SMOVL C00195 BC00195 V=166.7  +MOVJ EC00195
SFTOF3D
MOVL C00196 BC00196 V=1000.0  +MOVJ EC00196 VJ=100.00
'EndPath S3470
'Path S4850
SFTOF3D
MOVL C00197 BC00197 V=666.7  +MOVJ EC00197 VJ=100.00
SMOVL C00198 BC00198 V=166.7  +MOVJ EC00198
SREFP 3 C00199 BC00199  +REFP EC00199
CALL JOB:SEARCH-R1-S13D
SET P071 P006
SFTON3D P071
SMOVL C00200 BC00200 V=166.7  +MOVJ EC00200
SREFP 3 C00201 BC00201  +REFP EC00201
CALL JOB:SEARCH-R1-S13D
SET P071 P006
SFTON3D P071
SMOVL C00202 BC00202 V=166.7  +MOVJ EC00202
SMOVL C00203 BC00203 V=166.7  +MOVJ EC00203
SREFP 3 C00204 BC00204  +REFP EC00204
CALL JOB:SEARCH-R1-S13D
SET P071 P006
SFTON3D P071
SMOVL C00205 BC00205 V=166.7  +MOVJ EC00205
MOVL C00206 BC00206 V=1000.0  +MOVJ EC00206 VJ=100.00
'EndPath S4850
'Path S4851
SFTOF3D
MOVJ C00207 BC00207 VJ=100.00  +MOVJ EC00207 VJ=100.00
'POMIAR_DOD_WZM_BOK
MOVL C00208 BC00208 V=666.7  +MOVJ EC00208 VJ=100.00
SMOVL C00209 BC00209 V=166.7  +MOVJ EC00209
SREFP 3 C00210 BC00210  +REFP EC00210
CALL JOB:SEARCH-R1-S13D
SET P080 P006
SFTON3D P080
SMOVL C00211 BC00211 V=166.7  +MOVJ EC00211
SREFP 3 C00212 BC00212  +REFP EC00212
CALL JOB:SEARCH-R1-S13D
SET P080 P006
SFTON3D P080
SMOVL C00213 BC00213 V=166.7  +MOVJ EC00213
MOVL C00214 BC00214 V=666.7  +MOVJ EC00214 VJ=100.00
SMOVL C00215 BC00215 V=166.7  +MOVJ EC00215
SREFP 3 C00216 BC00216  +REFP EC00216
CALL JOB:SEARCH-R1-S13D
SET P042 P006
SFTON3D P042
SMOVL C00217 BC00217 V=166.7  +MOVJ EC00217
SREFP 3 C00218 BC00218  +REFP EC00218
CALL JOB:SEARCH-R1-S13D
SET P042 P006
SFTON3D P042
SMOVL C00219 BC00219 V=166.7  +MOVJ EC00219
SREFP 3 C00220 BC00220  +REFP EC00220
CALL JOB:SEARCH-R1-S13D
SET P043 P006
SFTON3D P043
SMOVL C00221 BC00221 V=166.7  +MOVJ EC00221
SREFP 3 C00222 BC00222  +REFP EC00222
CALL JOB:SEARCH-R1-S13D
SET P043 P006
SFTON3D P043
SMOVL C00223 BC00223 V=166.7  +MOVJ EC00223
SMOVL C00224 BC00224 V=1000.0  +MOVJ EC00224
MOVL C00225 BC00225 V=666.7  +MOVJ EC00225 VJ=100.00
SMOVL C00226 BC00226 V=166.7  +MOVJ EC00226
SREFP 3 C00227 BC00227  +REFP EC00227
CALL JOB:SEARCH-R1-S13D
SET P044 P006
SFTON3D P044
SMOVL C00228 BC00228 V=166.7  +MOVJ EC00228
SREFP 3 C00229 BC00229  +REFP EC00229
CALL JOB:SEARCH-R1-S13D
SET P044 P006
SFTON3D P044
SMOVL C00230 BC00230 V=166.7  +MOVJ EC00230
MOVL C00231 BC00231 V=666.7  +MOVJ EC00231 VJ=100.00
SMOVL C00232 BC00232 V=166.7  +MOVJ EC00232
SREFP 3 C00233 BC00233  +REFP EC00233
CALL JOB:SEARCH-R1-S13D
SET P045 P006
SFTON3D P045
SMOVL C00234 BC00234 V=166.7  +MOVJ EC00234
SREFP 3 C00235 BC00235  +REFP EC00235
CALL JOB:SEARCH-R1-S13D
SET P045 P006
SFTON3D P045
SMOVL C00236 BC00236 V=166.7  +MOVJ EC00236
SREFP 3 C00237 BC00237  +REFP EC00237
CALL JOB:SEARCH-R1-S13D
SET P046 P006
SFTON3D P046
SMOVL C00238 BC00238 V=166.7  +MOVJ EC00238
SREFP 3 C00239 BC00239  +REFP EC00239
CALL JOB:SEARCH-R1-S13D
SET P046 P006
SFTON3D P046
SMOVL C00240 BC00240 V=166.7  +MOVJ EC00240
SFTOF3D
SFTOF3D
MOVJ C00241 BC00241 VJ=100.00  +MOVJ EC00241 VJ=100.00
MOVL C00242 BC00242 V=666.7  +MOVJ EC00242 VJ=100.00
MOVL C00243 BC00243 V=1000.0  +MOVJ EC00243 VJ=0.78
SMOVL C00244 BC00244 V=166.7  +MOVJ EC00244
SREFP 3 C00245 BC00245  +REFP EC00245
CALL JOB:SEARCH-R1-S13D
SET P072 P006
SFTON3D P072
SMOVL C00246 BC00246 V=166.7  +MOVJ EC00246
SREFP 3 C00247 BC00247  +REFP EC00247
CALL JOB:SEARCH-R1-S13D
SET P072 P006
SFTON3D P072
SMOVL C00248 BC00248 V=166.7  +MOVJ EC00248
SMOVL C00249 BC00249 V=166.7  +MOVJ EC00249
SREFP 3 C00250 BC00250  +REFP EC00250
CALL JOB:SEARCH-R1-S13D
SET P072 P006
SFTON3D P072
SMOVL C00251 BC00251 V=166.7  +MOVJ EC00251
SFTOF3D
MOVL C00252 BC00252 V=1000.0  +MOVJ EC00252 VJ=100.00
'EndPath S4851
MOVJ C00253 BC00253 VJ=100.00  +MOVJ EC00253 VJ=100.00
MOVJ C00254 BC00254 VJ=100.00  +MOVJ EC00254 VJ=100.00
'Path S4852
SFTOF3D
MOVJ C00255 BC00255 VJ=100.00  +MOVJ EC00255 VJ=100.00
MOVL C00256 BC00256 V=666.7  +MOVJ EC00256 VJ=100.00
SMOVL C00257 BC00257 V=166.7  +MOVJ EC00257
SREFP 3 C00258 BC00258  +REFP EC00258
CALL JOB:SEARCH-R1-S13D
SET P073 P006
SFTON3D P073
SMOVL C00259 BC00259 V=166.7  +MOVJ EC00259
SMOVL C00260 BC00260 V=166.7  +MOVJ EC00260
SREFP 3 C00261 BC00261  +REFP EC00261
CALL JOB:SEARCH-R1-S13D
SET P073 P006
SFTON3D P073
SMOVL C00262 BC00262 V=166.7  +MOVJ EC00262
SMOVL C00263 BC00263 V=166.7  +MOVJ EC00263
SREFP 3 C00264 BC00264  +REFP EC00264
CALL JOB:SEARCH-R1-S13D
SET P073 P006
SFTON3D P073
SMOVL C00265 BC00265 V=166.7  +MOVJ EC00265
MOVL C00266 BC00266 V=1000.0  +MOVJ EC00266 VJ=100.00
'EndPath S4852
MOVJ C00267 BC00267 VJ=100.00  +MOVJ EC00267 VJ=100.00
'Path S4853
SFTOF3D
MOVJ C00268 BC00268 VJ=100.00  +MOVJ EC00268 VJ=100.00
MOVL C00269 BC00269 V=666.7  +MOVJ EC00269 VJ=100.00
SMOVL C00270 BC00270 V=166.7  +MOVJ EC00270
SREFP 3 C00271 BC00271  +REFP EC00271
CALL JOB:SEARCH-R1-S13D
SET P074 P006
SFTON3D P074
SMOVL C00272 BC00272 V=166.7  +MOVJ EC00272
SMOVL C00273 BC00273 V=333.3  +MOVJ EC00273
SREFP 3 C00274 BC00274  +REFP EC00274
CALL JOB:SEARCH-R1-S13D
SET P074 P006
SFTON3D P074
SMOVL C00275 BC00275 V=166.7  +MOVJ EC00275
SREFP 3 C00276 BC00276  +REFP EC00276
CALL JOB:SEARCH-R1-S13D
SET P074 P006
SFTON3D P074
SMOVL C00277 BC00277 V=166.7  +MOVJ EC00277
SFTOF3D
MOVL C00278 BC00278 V=1000.0  +MOVJ EC00278 VJ=100.00
'EndPath S4853
'Path S3467
SFTOF3D
MOVJ C00279 BC00279 VJ=100.00  +MOVJ EC00279 VJ=100.00
MOVJ C00280 BC00280 VJ=100.00  +MOVJ EC00280 VJ=100.00
MOVL C00281 BC00281 V=666.7  +MOVJ EC00281 VJ=100.00
SMOVL C00282 BC00282 V=166.7  +MOVJ EC00282
SREFP 3 C00283 BC00283  +REFP EC00283
CALL JOB:SEARCH-R1-S13D
SET P081 P006
SFTON3D P081
SMOVL C00284 BC00284 V=166.7  +MOVJ EC00284
SMOVL C00285 BC00285 V=166.7  +MOVJ EC00285
SREFP 3 C00286 BC00286  +REFP EC00286
CALL JOB:SEARCH-R1-S13D
SET P081 P006
SFTON3D P081
SMOVL C00287 BC00287 V=166.7  +MOVJ EC00287
SMOVL C00288 BC00288 V=800.0  +MOVJ EC00288
SMOVL C00289 BC00289 V=166.7  +MOVJ EC00289
SREFP 3 C00290 BC00290  +REFP EC00290
CALL JOB:SEARCH-R1-S13D
SET P081 P006
SFTON3D P081
SMOVL C00291 BC00291 V=166.7  +MOVJ EC00291
MOVJ C00292 BC00292 VJ=100.00  +MOVJ EC00292 VJ=100.00
MOVJ C00293 BC00293 VJ=100.00  +MOVJ EC00293 VJ=100.00
SFTOF3D
MOVJ C00294 BC00294 VJ=100.00  +MOVJ EC00294 VJ=100.00
MOVL C00295 BC00295 V=666.7  +MOVJ EC00295 VJ=100.00
SMOVL C00296 BC00296 V=166.7  +MOVJ EC00296
SREFP 3 C00297 BC00297  +REFP EC00297
CALL JOB:SEARCH-R1-S13D
SET P026 P006
SFTON3D P026
SMOVL C00298 BC00298 V=166.7  +MOVJ EC00298
SREFP 3 C00299 BC00299  +REFP EC00299
CALL JOB:SEARCH-R1-S13D
SET P026 P006
SFTON3D P026
SMOVL C00300 BC00300 V=166.7  +MOVJ EC00300
SMOVL C00301 BC00301 V=800.0  +MOVJ EC00301
SMOVL C00302 BC00302 V=166.7  +MOVJ EC00302
SREFP 3 C00303 BC00303  +REFP EC00303
CALL JOB:SEARCH-R1-S13D
SET P026 P006
SFTON3D P026
SMOVL C00304 BC00304 V=166.7  +MOVJ EC00304
MOVL C00305 BC00305 V=1000.0  +MOVJ EC00305 VJ=100.00
'EndPath S3467
MOVJ C00306 BC00306 VJ=100.00  +MOVJ EC00306 VJ=100.00
'Path S3466
SFTOF3D
MOVJ C00307 BC00307 VJ=100.00  +MOVJ EC00307 VJ=100.00
MOVL C00308 BC00308 V=666.7  +MOVJ EC00308 VJ=100.00
SMOVL C00309 BC00309 V=166.7  +MOVJ EC00309
SREFP 3 C00310 BC00310  +REFP EC00310
CALL JOB:SEARCH-R1-S13D
SET P025 P006
SFTON3D P025
SMOVL C00311 BC00311 V=166.7  +MOVJ EC00311
SMOVL C00312 BC00312 V=166.7  +MOVJ EC00312
SREFP 3 C00313 BC00313  +REFP EC00313
CALL JOB:SEARCH-R1-S13D
SET P025 P006
SFTON3D P025
SMOVL C00314 BC00314 V=166.7  +MOVJ EC00314
SMOVL C00315 BC00315 V=200.0  +MOVJ EC00315
SMOVL C00316 BC00316 V=166.7  +MOVJ EC00316
SREFP 3 C00317 BC00317  +REFP EC00317
CALL JOB:SEARCH-R1-S13D
SET P025 P006
SFTON3D P025
SMOVL C00318 BC00318 V=166.7  +MOVJ EC00318
MOVL C00319 BC00319 V=1000.0  +MOVJ EC00319 VJ=100.00
MOVL C00320 BC00320 V=1000.0  +MOVJ EC00320 VJ=0.78
SMOVL C00321 BC00321 V=166.7  +MOVJ EC00321
SREFP 3 C00322 BC00322  +REFP EC00322
CALL JOB:SEARCH-R1-S13D
SET P047 P006
SFTON3D P047
SMOVL C00323 BC00323 V=166.7  +MOVJ EC00323
SMOVL C00324 BC00324 V=166.7  +MOVJ EC00324
SREFP 3 C00325 BC00325  +REFP EC00325
CALL JOB:SEARCH-R1-S13D
SET P047 P006
SFTON3D P047
SMOVL C00326 BC00326 V=166.7  +MOVJ EC00326
MOVL C00327 BC00327 V=1000.0  +MOVJ EC00327 VJ=0.78
SMOVL C00328 BC00328 V=166.7  +MOVJ EC00328
SREFP 3 C00329 BC00329  +REFP EC00329
CALL JOB:SEARCH-R1-S13D
SET P048 P006
SFTON3D P048
SMOVL C00330 BC00330 V=166.7  +MOVJ EC00330
SMOVL C00331 BC00331 V=166.7  +MOVJ EC00331
SREFP 3 C00332 BC00332  +REFP EC00332
CALL JOB:SEARCH-R1-S13D
SET P048 P006
SFTON3D P048
SMOVL C00333 BC00333 V=166.7  +MOVJ EC00333
SFTOF3D
MOVL C00334 BC00334 V=1000.0  +MOVJ EC00334 VJ=0.78
'EndPath S3466
MOVJ C00335 BC00335 VJ=100.00  +MOVJ EC00335 VJ=100.00
'Path S3469
SFTOF3D
MOVJ C00336 BC00336 VJ=100.00  +MOVJ EC00336 VJ=100.00
MOVL C00337 BC00337 V=666.7  +MOVJ EC00337 VJ=100.00
SMOVL C00338 BC00338 V=166.7  +MOVJ EC00338
SREFP 3 C00339 BC00339  +REFP EC00339
CALL JOB:SEARCH-R1-S13D
SET P055 P006
SFTON3D P055
SMOVL C00340 BC00340 V=166.7  +MOVJ EC00340
SREFP 3 C00341 BC00341  +REFP EC00341
CALL JOB:SEARCH-R1-S13D
SET P055 P006
SFTON3D P055
SMOVL C00342 BC00342 V=166.7  +MOVJ EC00342
MOVL C00343 BC00343 V=666.7  +MOVJ EC00343 VJ=100.00
SMOVL C00344 BC00344 V=166.7  +MOVJ EC00344
SREFP 3 C00345 BC00345  +REFP EC00345
CALL JOB:SEARCH-R1-S13D
SET P049 P006
SFTON3D P049
SMOVL C00346 BC00346 V=166.7  +MOVJ EC00346
SREFP 3 C00347 BC00347  +REFP EC00347
CALL JOB:SEARCH-R1-S13D
SET P049 P006
SFTON3D P049
SMOVL C00348 BC00348 V=166.7  +MOVJ EC00348
MOVL C00349 BC00349 V=666.7  +MOVJ EC00349 VJ=100.00
SMOVL C00350 BC00350 V=166.7  +MOVJ EC00350
SREFP 3 C00351 BC00351  +REFP EC00351
CALL JOB:SEARCH-R1-S13D
SET P028 P006
SFTON3D P028
SMOVL C00352 BC00352 V=166.7  +MOVJ EC00352
SREFP 3 C00353 BC00353  +REFP EC00353
CALL JOB:SEARCH-R1-S13D
SET P028 P006
SFTON3D P028
SMOVL C00354 BC00354 V=166.7  +MOVJ EC00354
SMOVL C00355 BC00355 V=333.3  +MOVJ EC00355
SMOVL C00356 BC00356 V=166.7  +MOVJ EC00356
SREFP 3 C00357 BC00357  +REFP EC00357
CALL JOB:SEARCH-R1-S13D
SET P028 P006
SFTON3D P028
SMOVL C00358 BC00358 V=166.7  +MOVJ EC00358
MOVL C00359 BC00359 V=1000.0  +MOVJ EC00359 VJ=100.00
'EndPath S3469
MOVJ C00360 BC00360 VJ=100.00  +MOVJ EC00360 VJ=100.00
'Path S3474
SFTOF3D
MOVJ C00361 BC00361 VJ=100.00  +MOVJ EC00361 VJ=100.00
MOVL C00362 BC00362 V=666.7  +MOVJ EC00362 VJ=100.00
SMOVL C00363 BC00363 V=166.7  +MOVJ EC00363
SREFP 3 C00364 BC00364  +REFP EC00364
CALL JOB:SEARCH-R1-S13D
SET P033 P006
SFTON3D P033
SMOVL C00365 BC00365 V=166.7  +MOVJ EC00365
SREFP 3 C00366 BC00366  +REFP EC00366
CALL JOB:SEARCH-R1-S13D
SET P033 P006
SFTON3D P033
SMOVL C00367 BC00367 V=166.7  +MOVJ EC00367
SMOVL C00368 BC00368 V=250.0  +MOVJ EC00368
SMOVL C00369 BC00369 V=166.7  +MOVJ EC00369
SREFP 3 C00370 BC00370  +REFP EC00370
CALL JOB:SEARCH-R1-S13D
SET P033 P006
SFTON3D P033
SMOVL C00371 BC00371 V=166.7  +MOVJ EC00371
MOVL C00372 BC00372 V=1000.0  +MOVJ EC00372 VJ=100.00
'EndPath S3474
'Path S3468
SFTOF3D
MOVJ C00373 BC00373 VJ=100.00  +MOVJ EC00373 VJ=100.00
MOVL C00374 BC00374 V=666.7  +MOVJ EC00374 VJ=100.00
SMOVL C00375 BC00375 V=166.7  +MOVJ EC00375
SREFP 3 C00376 BC00376  +REFP EC00376
CALL JOB:SEARCH-R1-S13D
SET P027 P006
SFTON3D P027
SMOVL C00377 BC00377 V=166.7  +MOVJ EC00377
SMOVL C00378 BC00378 V=166.7  +MOVJ EC00378
SREFP 3 C00379 BC00379  +REFP EC00379
CALL JOB:SEARCH-R1-S13D
SET P027 P006
SFTON3D P027
SMOVL C00380 BC00380 V=166.7  +MOVJ EC00380
SMOVL C00381 BC00381 V=166.7  +MOVJ EC00381
SREFP 3 C00382 BC00382  +REFP EC00382
CALL JOB:SEARCH-R1-S13D
SET P027 P006
SFTON3D P027
SMOVL C00383 BC00383 V=166.7  +MOVJ EC00383
MOVL C00384 BC00384 V=1000.0  +MOVJ EC00384 VJ=100.00
'EndPath S3468
'Path S3471
SFTOF3D
MOVJ C00385 BC00385 VJ=100.00  +MOVJ EC00385 VJ=100.00
MOVL C00386 BC00386 V=666.7  +MOVJ EC00386 VJ=100.00
SMOVL C00387 BC00387 V=166.7  +MOVJ EC00387
SREFP 3 C00388 BC00388  +REFP EC00388
CALL JOB:SEARCH-R1-S13D
SET P030 P006
SFTON3D P030
SMOVL C00389 BC00389 V=166.7  +MOVJ EC00389
SREFP 3 C00390 BC00390  +REFP EC00390
CALL JOB:SEARCH-R1-S13D
SET P030 P006
SFTON3D P030
SMOVL C00391 BC00391 V=166.7  +MOVJ EC00391
MOVL C00392 BC00392 V=1000.0  +MOVJ EC00392 VJ=100.00
'EndPath S3471
'Path S3472
SFTOF3D
MOVJ C00393 BC00393 VJ=100.00  +MOVJ EC00393 VJ=100.00
MOVL C00394 BC00394 V=666.7  +MOVJ EC00394 VJ=100.00
SMOVL C00395 BC00395 V=166.7  +MOVJ EC00395
SREFP 3 C00396 BC00396  +REFP EC00396
CALL JOB:SEARCH-R1-S13D
SET P031 P006
SFTON3D P031
SMOVL C00397 BC00397 V=166.7  +MOVJ EC00397
SREFP 3 C00398 BC00398  +REFP EC00398
CALL JOB:SEARCH-R1-S13D
SET P031 P006
SFTON3D P031
SMOVL C00399 BC00399 V=166.7  +MOVJ EC00399
MOVL C00400 BC00400 V=1000.0  +MOVJ EC00400 VJ=100.00
MOVL C00401 BC00401 V=666.7  +MOVJ EC00401 VJ=100.00
SMOVL C00402 BC00402 V=166.7  +MOVJ EC00402
SREFP 3 C00403 BC00403  +REFP EC00403
CALL JOB:SEARCH-R1-S13D
SET P098 P006
SFTON3D P098
SMOVL C00404 BC00404 V=166.7  +MOVJ EC00404
SREFP 3 C00405 BC00405  +REFP EC00405
CALL JOB:SEARCH-R1-S13D
SET P098 P006
SFTON3D P098
SMOVL C00406 BC00406 V=166.7  +MOVJ EC00406
MOVL C00407 BC00407 V=1000.0  +MOVJ EC00407 VJ=100.00
'EndPath S3472
MOVJ C00408 BC00408 VJ=100.00  +MOVJ EC00408 VJ=100.00
'Path S3472
SFTOF3D
MOVJ C00409 BC00409 VJ=100.00  +MOVJ EC00409 VJ=100.00
MOVL C00410 BC00410 V=666.7  +MOVJ EC00410 VJ=100.00
SMOVL C00411 BC00411 V=166.7  +MOVJ EC00411
SREFP 3 C00412 BC00412  +REFP EC00412
CALL JOB:SEARCH-R1-S13D
SET P032 P006
SFTON3D P032
SMOVL C00413 BC00413 V=166.7  +MOVJ EC00413
SREFP 3 C00414 BC00414  +REFP EC00414
CALL JOB:SEARCH-R1-S13D
SET P032 P006
SFTON3D P032
SMOVL C00415 BC00415 V=166.7  +MOVJ EC00415
SMOVL C00416 BC00416 V=133.3  +MOVJ EC00416
SREFP 3 C00417 BC00417  +REFP EC00417
CALL JOB:SEARCH-R1-S13D
SET P032 P006
SFTON3D P032
SMOVL C00418 BC00418 V=166.7  +MOVJ EC00418
MOVL C00419 BC00419 V=1000.0  +MOVJ EC00419 VJ=100.00
'EndPath S3472
MOVJ C00420 BC00420 VJ=100.00  +MOVJ EC00420 VJ=100.00
'Path S3477
SFTOF3D
MOVJ C00421 BC00421 VJ=100.00  +MOVJ EC00421 VJ=100.00
SMOVL C00422 BC00422 V=166.7  +MOVJ EC00422
SREFP 3 C00423 BC00423  +REFP EC00423
CALL JOB:SEARCH-R1-S13D
SET P069 P006
SFTON3D P069
SMOVL C00424 BC00424 V=250.0  +MOVJ EC00424
SMOVL C00425 BC00425 V=250.0  +MOVJ EC00425
SMOVL C00426 BC00426 V=166.7  +MOVJ EC00426
SREFP 3 C00427 BC00427  +REFP EC00427
CALL JOB:SEARCH-R1-S13D
SET P069 P006
SFTON3D P069
SMOVL C00428 BC00428 V=166.7  +MOVJ EC00428
SFTOF3D
SMOVL C00429 BC00429 V=666.7  +MOVJ EC00429
MOVL C00430 BC00430 V=666.7  +MOVJ EC00430 VJ=100.00
SMOVL C00431 BC00431 V=166.7  +MOVJ EC00431
SREFP 3 C00432 BC00432  +REFP EC00432
CALL JOB:SEARCH-R1-S13D
SET P052 P006
SFTON3D P052
SMOVL C00433 BC00433 V=166.7  +MOVJ EC00433
SREFP 3 C00434 BC00434  +REFP EC00434
CALL JOB:SEARCH-R1-S13D
SET P052 P006
SFTON3D P052
SMOVL C00435 BC00435 V=166.7  +MOVJ EC00435
MOVL C00436 BC00436 V=1000.0  +MOVJ EC00436 VJ=100.00
'EndPath S3477
MOVJ C00437 BC00437 VJ=100.00  +MOVJ EC00437 VJ=100.00
'poprawi searcha- nie mialem
'wyciecia
'Path S3478
SFTOF3D
MOVJ C00438 BC00438 VJ=100.00  +MOVJ EC00438 VJ=100.00
MOVL C00439 BC00439 V=666.7  +MOVJ EC00439 VJ=100.00
SMOVL C00440 BC00440 V=166.7  +MOVJ EC00440
SREFP 3 C00441 BC00441  +REFP EC00441
CALL JOB:SEARCH-R1-S13D
SET P053 P006
SFTON3D P053
SMOVL C00442 BC00442 V=166.7  +MOVJ EC00442
SREFP 3 C00443 BC00443  +REFP EC00443
CALL JOB:SEARCH-R1-S13D
SET P053 P006
SFTON3D P053
SMOVL C00444 BC00444 V=166.7  +MOVJ EC00444
MOVL C00445 BC00445 V=1000.0  +MOVJ EC00445 VJ=100.00
'EndPath S3478
'
MOVJ C00446 BC00446 VJ=100.00  +MOVJ EC00446 VJ=100.00
'Path W3476
SFTOF3D
SFTON3D P033
MOVJ C00447 BC00447 VJ=100.00  +MOVJ EC00447 VJ=100.00
SMOVL C00448 BC00448 V=800.0  +MOVJ EC00448
SMOVL C00449 BC00449 V=166.7 PL=0  +MOVJ EC00449
MACRO1 MJ#(0) ARGF14
ARCON
SMOVL C00450 BC00450 V=10.0  +MOVJ EC00450
ARCOF
SMOVL C00451 BC00451 V=800.0  +MOVJ EC00451
SMOVL C00452 BC00452 V=1000.0  +MOVJ EC00452
SFTOF3D
'EndPath W3476
'Path W3477
SFTOF3D
SFTON3D P033
MOVJ C00453 BC00453 VJ=100.00  +MOVJ EC00453 VJ=100.00
SMOVL C00454 BC00454 V=800.0  +MOVJ EC00454
SMOVL C00455 BC00455 V=166.7 PL=0  +MOVJ EC00455
SMOVL C00456 BC00456 V=10.0  +MOVJ EC00456
SMOVL C00457 BC00457 V=10.0  +MOVJ EC00457
SMOVL C00458 BC00458 V=10.0  +MOVJ EC00458
ARCOF
SMOVL C00459 BC00459 V=800.0  +MOVJ EC00459
SMOVL C00460 BC00460 V=1000.0  +MOVJ EC00460
SFTOF3D
'EndPath W3477
MOVJ C00461 BC00461 VJ=100.00  +MOVJ EC00461 VJ=100.00
'Path W3478
SFTOF3D
SFTON3D P033
MOVJ C00462 BC00462 VJ=100.00  +MOVJ EC00462 VJ=100.00
SMOVL C00463 BC00463 V=800.0  +MOVJ EC00463
SMOVL C00464 BC00464 V=166.7 PL=0  +MOVJ EC00464
ARCON
SMOVL C00465 BC00465 V=10.0  +MOVJ EC00465
SMOVL C00466 BC00466 V=10.0  +MOVJ EC00466
SMOVL C00467 BC00467 V=10.0  +MOVJ EC00467
ARCOF
SMOVL C00468 BC00468 V=800.0  +MOVJ EC00468
SMOVL C00469 BC00469 V=1000.0  +MOVJ EC00469
SFTOF3D
'EndPath W3478
MOVJ C00470 BC00470 VJ=100.00  +MOVJ EC00470 VJ=100.00
MOVJ C00471 BC00471 VJ=100.00  +MOVJ EC00471 VJ=100.00
SFTOF3D
SFTON3D P081
MOVJ C00472 BC00472 VJ=100.00  +MOVJ EC00472 VJ=100.00
SMOVL C00473 BC00473 V=800.0  +MOVJ EC00473
SMOVL C00474 BC00474 V=166.7 PL=0  +MOVJ EC00474
ARCON
SMOVL C00475 BC00475 V=9.2  +MOVJ EC00475
ARCOF
SMOVL C00476 BC00476 V=800.0  +MOVJ EC00476
SMOVL C00477 BC00477 V=1000.0  +MOVJ EC00477
SFTOF3D
'EndPath W3479
'Path W3480
SFTOF3D
SFTON3D P081
MOVJ C00478 BC00478 VJ=100.00  +MOVJ EC00478 VJ=100.00
SMOVL C00479 BC00479 V=800.0  +MOVJ EC00479
SMOVL C00480 BC00480 V=150.0 PL=0  +MOVJ EC00480
ARCON
SMOVL C00481 BC00481 V=10.0  +MOVJ EC00481
ARCOF
SMOVL C00482 BC00482 V=800.0  +MOVJ EC00482
SMOVL C00483 BC00483 V=1000.0  +MOVJ EC00483
SFTOF3D
'EndPath W3480
'Path W3481
SFTOF3D
SFTON3D P081
MOVJ C00484 BC00484 VJ=100.00  +MOVJ EC00484 VJ=100.00
SMOVL C00485 BC00485 V=800.0  +MOVJ EC00485
SMOVL C00486 BC00486 V=150.0 PL=0  +MOVJ EC00486
ARCON
SMOVL C00487 BC00487 V=10.0  +MOVJ EC00487
ARCOF
SMOVL C00488 BC00488 V=800.0  +MOVJ EC00488
SMOVL C00489 BC00489 V=1000.0  +MOVJ EC00489
SFTOF3D
'EndPath W3481
MOVJ C00490 BC00490 VJ=100.00  +MOVJ EC00490 VJ=100.00
'uwaga na podajnik
'Path W3481
SFTOF3D
SFTON3D P081
MOVJ C00491 BC00491 VJ=50.00  +MOVJ EC00491 VJ=15.00
SMOVL C00492 BC00492 V=800.0  +MOVJ EC00492
SMOVL C00493 BC00493 V=150.0 PL=0  +MOVJ EC00493
ARCON
SMOVL C00494 BC00494 V=10.0  +MOVJ EC00494
ARCOF
SMOVL C00495 BC00495 V=800.0  +MOVJ EC00495
SMOVL C00496 BC00496 V=1000.0  +MOVJ EC00496
SFTOF3D
'9
'Path W3479
MOVJ C00497 BC00497 VJ=100.00  +MOVJ EC00497 VJ=100.00
SFTOF3D
SFTON3D P026
MOVJ C00498 BC00498 VJ=100.00  +MOVJ EC00498 VJ=100.00
SMOVL C00499 BC00499 V=800.0  +MOVJ EC00499
SMOVL C00500 BC00500 V=166.7 PL=0  +MOVJ EC00500
ARCON
SMOVL C00501 BC00501 V=9.2  +MOVJ EC00501
SMOVL C00502 BC00502 V=9.2  +MOVJ EC00502
SMOVL C00503 BC00503 V=9.2  +MOVJ EC00503
ARCOF
SMOVL C00504 BC00504 V=800.0  +MOVJ EC00504
SMOVL C00505 BC00505 V=1000.0  +MOVJ EC00505
SFTOF3D
'EndPath W3479
'Path W3480
SFTOF3D
SFTON3D P026
MOVJ C00506 BC00506 VJ=100.00  +MOVJ EC00506 VJ=100.00
SMOVL C00507 BC00507 V=800.0  +MOVJ EC00507
SMOVL C00508 BC00508 V=150.0 PL=0  +MOVJ EC00508
ARCON
SMOVL C00509 BC00509 V=10.0  +MOVJ EC00509
SMOVL C00510 BC00510 V=10.0  +MOVJ EC00510
SMOVL C00511 BC00511 V=10.0  +MOVJ EC00511
ARCOF
SMOVL C00512 BC00512 V=800.0  +MOVJ EC00512
SMOVL C00513 BC00513 V=1000.0  +MOVJ EC00513
SFTOF3D
'EndPath W3480
'Path W3481
SFTOF3D
SFTON3D P026
MOVJ C00514 BC00514 VJ=100.00  +MOVJ EC00514 VJ=100.00
SMOVL C00515 BC00515 V=800.0  +MOVJ EC00515
SMOVL C00516 BC00516 V=150.0 PL=0  +MOVJ EC00516
ARCON
SMOVL C00517 BC00517 V=10.0  +MOVJ EC00517
ARCOF
SMOVL C00518 BC00518 V=800.0  +MOVJ EC00518
SMOVL C00519 BC00519 V=1000.0  +MOVJ EC00519
SFTOF3D
'EndPath W3481
MOVJ C00520 BC00520 VJ=100.00  +MOVJ EC00520 VJ=100.00
'uwaga na podajnik
'Path W3481
SFTOF3D
SFTON3D P026
MOVJ C00521 BC00521 VJ=50.00  +MOVJ EC00521 VJ=15.00
SMOVL C00522 BC00522 V=800.0  +MOVJ EC00522
SMOVL C00523 BC00523 V=150.0 PL=0  +MOVJ EC00523
ARCON
SMOVL C00524 BC00524 V=10.0  +MOVJ EC00524
SMOVL C00525 BC00525 V=10.0  +MOVJ EC00525
ARCOF
SMOVL C00526 BC00526 V=800.0  +MOVJ EC00526
SMOVL C00527 BC00527 V=1000.0  +MOVJ EC00527
SFTOF3D
'EndPath W3481
'brak dostepu offset drutu 1cm
'Path W3482
SFTOF3D
SFTON3D P026
MOVJ C00528 BC00528 VJ=100.00  +MOVJ EC00528 VJ=100.00
SMOVL C00529 BC00529 V=800.0  +MOVJ EC00529
SMOVL C00530 BC00530 V=150.0 PL=0  +MOVJ EC00530
ARCON
SMOVL C00531 BC00531 V=10.0  +MOVJ EC00531
ARCOF
SMOVL C00532 BC00532 V=800.0  +MOVJ EC00532
SMOVL C00533 BC00533 V=1000.0  +MOVJ EC00533
SFTOF3D
'EndPath W3482
MOVJ C00534 BC00534 VJ=100.00  +MOVJ EC00534 VJ=100.00
MOVJ C00535 BC00535 VJ=100.00  +MOVJ EC00535 VJ=100.00
'10
'11
'Path W3484
SFTOF3D
SFTON3D P048
MOVJ C00536 BC00536 VJ=100.00  +MOVJ EC00536 VJ=100.00
SMOVL C00537 BC00537 V=800.0  +MOVJ EC00537
SMOVL C00538 BC00538 V=150.0 PL=0  +MOVJ EC00538
ARCON
SWVON WEV#(16)
SMOVL C00539 BC00539 V=10.0  +MOVJ EC00539
SMOVL C00540 BC00540 V=10.0  +MOVJ EC00540
SMOVL C00541 BC00541 V=10.0  +MOVJ EC00541
SFTON3D P047
SMOVL C00542 BC00542 V=10.0  +MOVJ EC00542
SMOVL C00543 BC00543 V=10.0  +MOVJ EC00543
SFTON3D P025
SMOVL C00544 BC00544 V=10.0  +MOVJ EC00544
SMOVL C00545 BC00545 V=10.0  +MOVJ EC00545
ARCOF
SWVOF
SMOVL C00546 BC00546 V=800.0  +MOVJ EC00546
SMOVL C00547 BC00547 V=1000.0  +MOVJ EC00547
SFTOF3D
'EndPath W3484
MOVJ C00548 BC00548 VJ=100.00  +MOVJ EC00548 VJ=100.00
'brak dostepu offset drutu 1cm
'Path W3483
SFTOF3D
SFTON3D P025
MOVJ C00549 BC00549 VJ=100.00  +MOVJ EC00549 VJ=100.00
SMOVL C00550 BC00550 V=800.0  +MOVJ EC00550
SMOVL C00551 BC00551 V=166.7 PL=0  +MOVJ EC00551
ARCON
SMOVL C00552 BC00552 V=10.0  +MOVJ EC00552
ARCOF
SMOVL C00553 BC00553 V=800.0  +MOVJ EC00553
SMOVL C00554 BC00554 V=1000.0  +MOVJ EC00554
SFTOF3D
'EndPath W3483
MOVJ C00555 BC00555 VJ=100.00  +MOVJ EC00555 VJ=100.00
MOVJ C00556 BC00556 VJ=100.00  +MOVJ EC00556 VJ=100.00
MOVJ C00557 BC00557 VJ=100.00  +MOVJ EC00557 VJ=100.00
'Path W4854
SFTOF3D
SFTON3D P073
MOVJ C00558 BC00558 VJ=100.00  +MOVJ EC00558 VJ=100.00
SMOVL C00559 BC00559 V=800.0  +MOVJ EC00559
SMOVL C00560 BC00560 V=150.0 PL=0  +MOVJ EC00560
MACRO1 MJ#(0) ARGF9
ARCON
SWVON WEV#(16)
SMOVL C00561 BC00561 V=7.5  +MOVJ EC00561
SFTON3D P074
SMOVL C00562 BC00562 V=7.5  +MOVJ EC00562
SMOVL C00563 BC00563 V=7.5  +MOVJ EC00563
ARCOF
SWVOF
SMOVL C00564 BC00564 V=800.0  +MOVJ EC00564
COMM MOVJ C00565 BC00565 VJ=50.00  +MOVJ EC00565 VJ=100.00
COMM SMOVL C00566 BC00566 V=166.7  +MOVJ EC00566
COMM SMOVL C00567 BC00567 V=166.7  +MOVJ EC00567
COMM SMOVL C00568 BC00568 V=50.0 PL=0  +MOVJ EC00568
COMM ARCON
COMM SMOVL C00569 BC00569 V=9.2  +MOVJ EC00569
COMM SMOVL C00570 BC00570 V=9.2  +MOVJ EC00570
COMM ARCOF
COMM SMOVL C00571 BC00571 V=1000.0  +MOVJ EC00571
SFTOF3D
'EndPath W4854
'12
MOVJ C00572 BC00572 VJ=100.00  +MOVJ EC00572 VJ=100.00
MOVJ C00573 BC00573 VJ=100.00  +MOVJ EC00573 VJ=100.00
MOVJ C00574 BC00574 VJ=100.00  +MOVJ EC00574 VJ=100.00
'Path W3485
SFTOF3D
SMOVL C00575 BC00575 V=1000.0  +MOVJ EC00575
SFTON3D P034
MOVJ C00576 BC00576 VJ=100.00  +MOVJ EC00576 VJ=100.00
SMOVL C00577 BC00577 V=800.0  +MOVJ EC00577
SMOVL C00578 BC00578 V=150.0 PL=0  +MOVJ EC00578
MACRO1 MJ#(0) ARGF14
ARCON
SMOVL C00579 BC00579 V=10.0  +MOVJ EC00579
SMOVL C00580 BC00580 V=10.0  +MOVJ EC00580
SMOVL C00581 BC00581 V=10.0  +MOVJ EC00581
ARCOF
SMOVL C00582 BC00582 V=800.0  +MOVJ EC00582
SMOVL C00583 BC00583 V=1000.0  +MOVJ EC00583
SFTOF3D
MOVJ C00584 BC00584 VJ=80.00  +MOVJ EC00584 VJ=80.00
MOVJ C00585 BC00585 VJ=80.00  +MOVJ EC00585 VJ=80.00
MOVJ C00586 BC00586 VJ=80.00  +MOVJ EC00586 VJ=80.00
MACRO1 MJ#(0) ARGF6
SFTON3D P063
SMOVL C00587 BC00587 V=166.7  +MOVJ EC00587
ARCON
SMOVL C00588 BC00588 V=11.7  +MOVJ EC00588
SMOVL C00589 BC00589 V=11.7  +MOVJ EC00589
SFTON3D P062
SMOVL C00590 BC00590 V=11.0  +MOVJ EC00590
SMOVL C00591 BC00591 V=11.0  +MOVJ EC00591
SFTON3D P061
SMOVL C00592 BC00592 V=11.0  +MOVJ EC00592
SMOVL C00593 BC00593 V=11.0  +MOVJ EC00593
ARCOF
SMOVL C00594 BC00594 V=800.0  +MOVJ EC00594
SFTOF3D
MOVJ C00595 BC00595 VJ=80.00  +MOVJ EC00595 VJ=80.00
MOVJ C00596 BC00596 VJ=80.00  +MOVJ EC00596 VJ=80.00
MOVJ C00597 BC00597 VJ=80.00  +MOVJ EC00597 VJ=80.00
'EndPath W3485
'Path W3486
SFTOF3D
SFTON3D P050
MOVJ C00598 BC00598 VJ=100.00  +MOVJ EC00598 VJ=100.00
SMOVL C00599 BC00599 V=800.0  +MOVJ EC00599
SMOVL C00600 BC00600 V=150.0 PL=0  +MOVJ EC00600
MACRO1 MJ#(0) ARGF14
ARCON
SMOVL C00601 BC00601 V=10.0  +MOVJ EC00601
SMOVL C00602 BC00602 V=10.0  +MOVJ EC00602
SMOVL C00603 BC00603 V=10.0  +MOVJ EC00603
ARCOF
SMOVL C00604 BC00604 V=800.0  +MOVJ EC00604
SMOVL C00605 BC00605 V=1000.0  +MOVJ EC00605
SFTOF3D
'EndPath W3486
MOVJ C00606 BC00606 VJ=100.00  +MOVJ EC00606 VJ=100.00
'Path W3485
SFTOF3D
SFTON3D P034
MOVJ C00607 BC00607 VJ=100.00  +MOVJ EC00607 VJ=100.00
SMOVL C00608 BC00608 V=800.0  +MOVJ EC00608
SMOVL C00609 BC00609 V=166.7 PL=0  +MOVJ EC00609
SREFP 1 C00610 BC00610  +REFP EC00610
SREFP 2 C00611 BC00611  +REFP EC00611
ARCON
SWVON WEV#(20)
SMOVL C00612 BC00612 V=9.2  +MOVJ EC00612
SMOVL C00613 BC00613 V=9.2  +MOVJ EC00613
SMOVL C00614 BC00614 V=9.2  +MOVJ EC00614
ARCOF
SWVOF
SMOVL C00615 BC00615 V=800.0  +MOVJ EC00615
SMOVL C00616 BC00616 V=1000.0  +MOVJ EC00616
SFTOF3D
'EndPath W3485
'Path W3487
SFTOF3D
SFTON3D P054
MOVJ C00617 BC00617 VJ=100.00  +MOVJ EC00617 VJ=100.00
SMOVL C00618 BC00618 V=800.0  +MOVJ EC00618
SMOVL C00619 BC00619 V=150.0 PL=0  +MOVJ EC00619
ARCON
SWVON WEV#(20)
SMOVL C00620 BC00620 V=9.2  +MOVJ EC00620
SMOVL C00621 BC00621 V=9.2  +MOVJ EC00621
SMOVL C00622 BC00622 V=9.2  +MOVJ EC00622
ARCOF
SWVOF
SMOVL C00623 BC00623 V=800.0  +MOVJ EC00623
SMOVL C00624 BC00624 V=1000.0  +MOVJ EC00624
SFTOF3D
'EndPath W3487
MOVJ C00625 BC00625 VJ=100.00  +MOVJ EC00625 VJ=100.00
'Path W3487
SFTOF3D
SFTON3D P028
MOVJ C00626 BC00626 VJ=100.00  +MOVJ EC00626 VJ=100.00
SMOVL C00627 BC00627 V=800.0  +MOVJ EC00627
SMOVL C00628 BC00628 V=150.0 PL=0  +MOVJ EC00628
ARCON
SWVON WEV#(16)
SMOVL C00629 BC00629 V=9.2  +MOVJ EC00629
SFTON3D P049
SMOVL C00630 BC00630 V=9.2  +MOVJ EC00630
SMOVL C00631 BC00631 V=9.2  +MOVJ EC00631
SFTON3D P055
SMOVL C00632 BC00632 V=9.2  +MOVJ EC00632
SMOVL C00633 BC00633 V=9.2  +MOVJ EC00633
ARCOF
SWVOF
SMOVL C00634 BC00634 V=800.0  +MOVJ EC00634
SMOVL C00635 BC00635 V=1000.0  +MOVJ EC00635
SFTOF3D
'EndPath W3487
MOVJ C00636 BC00636 VJ=100.00  +MOVJ EC00636 VJ=100.00
MOVJ C00637 BC00637 VJ=100.00  +MOVJ EC00637 VJ=100.00
'brak dostepu offset 5mm
'Path W3488
SFTOF3D
SFTON3D P028
MOVJ C00638 BC00638 VJ=100.00  +MOVJ EC00638 VJ=100.00
SMOVL C00639 BC00639 V=800.0  +MOVJ EC00639
SMOVL C00640 BC00640 V=150.0 PL=0  +MOVJ EC00640
ARCON
SMOVL C00641 BC00641 V=11.7  +MOVJ EC00641
ARCOF
SMOVL C00642 BC00642 V=800.0  +MOVJ EC00642
SMOVL C00643 BC00643 V=1000.0  +MOVJ EC00643
SFTOF3D
'EndPath W3488
MOVJ C00644 BC00644 VJ=100.00  +MOVJ EC00644 VJ=100.00
'13
'Path W3489
SFTOF3D
SFTON3D P030
MOVJ C00645 BC00645 VJ=100.00  +MOVJ EC00645 VJ=100.00
SMOVL C00646 BC00646 V=800.0  +MOVJ EC00646
SMOVL C00647 BC00647 V=150.0 PL=0  +MOVJ EC00647
MACRO1 MJ#(0) ARGF9
ARCON
SWVON WEV#(10)
SFTON3D P031
SMOVL C00648 BC00648 V=6.7  +MOVJ EC00648
SFTON3D P098
SMOVL C00649 BC00649 V=6.7  +MOVJ EC00649
ARCOF
SWVOF
SMOVL C00650 BC00650 V=800.0  +MOVJ EC00650
SMOVL C00651 BC00651 V=1000.0  +MOVJ EC00651
SFTOF3D
'EndPath W3489
'Path W3490
SFTOF3D
MOVJ C00652 BC00652 VJ=100.00  +MOVJ EC00652 VJ=100.00
MACRO1 MJ#(0) ARGF6
SFTON3D P069
SMOVL C00653 BC00653 V=250.0  +MOVJ EC00653
ARCON
SMOVL C00654 BC00654 V=11.7  +MOVJ EC00654
ARCOF
SMOVL C00655 BC00655 V=250.0  +MOVJ EC00655
SFTOF3D
SFTON3D P052
MOVJ C00656 BC00656 VJ=100.00  +MOVJ EC00656 VJ=100.00
SMOVL C00657 BC00657 V=800.0  +MOVJ EC00657
SMOVL C00658 BC00658 V=150.0 PL=0  +MOVJ EC00658
MACRO1 MJ#(0) ARGF14
ARCON
SMOVL C00659 BC00659 V=10.0  +MOVJ EC00659
SMOVL C00660 BC00660 V=10.0  +MOVJ EC00660
SMOVL C00661 BC00661 V=10.0  +MOVJ EC00661
ARCOF
SMOVL C00662 BC00662 V=800.0  +MOVJ EC00662
SMOVL C00663 BC00663 V=1000.0  +MOVJ EC00663
SFTOF3D
'EndPath W3490
MOVJ C00664 BC00664 VJ=100.00  +MOVJ EC00664 VJ=100.00
'poprawic spoine - nie mialem w
'yciecia
'Path W3491
SFTOF3D
SFTON3D P053
MOVJ C00665 BC00665 VJ=100.00  +MOVJ EC00665 VJ=100.00
SMOVL C00666 BC00666 V=800.0  +MOVJ EC00666
SMOVL C00667 BC00667 V=150.0 PL=0  +MOVJ EC00667
ARCON
SMOVL C00668 BC00668 V=10.0  +MOVJ EC00668
SMOVL C00669 BC00669 V=10.0  +MOVJ EC00669
SMOVL C00670 BC00670 V=10.0  +MOVJ EC00670
ARCOF
SMOVL C00671 BC00671 V=800.0  +MOVJ EC00671
SMOVL C00672 BC00672 V=1000.0  +MOVJ EC00672
SFTOF3D
'EndPath W3491
'14
'15-brak
MOVJ C00673 BC00673 VJ=100.00  +MOVJ EC00673 VJ=100.00
'16
'Path W3491
SFTOF3D
SFTON3D P029
MOVJ C00674 BC00674 VJ=100.00  +MOVJ EC00674 VJ=100.00
SMOVL C00675 BC00675 V=800.0  +MOVJ EC00675
SMOVL C00676 BC00676 V=150.0 PL=0  +MOVJ EC00676
ARCON
SMOVL C00677 BC00677 V=10.0  +MOVJ EC00677
SFTON3D P039
SMOVL C00678 BC00678 V=10.0  +MOVJ EC00678
SMOVL C00679 BC00679 V=10.0  +MOVJ EC00679
ARCOF
SMOVL C00680 BC00680 V=800.0  +MOVJ EC00680
SMOVL C00681 BC00681 V=1000.0  +MOVJ EC00681
SFTOF3D
'EndPath W3491
MOVJ C00682 BC00682 VJ=100.00  +MOVJ EC00682 VJ=100.00
'Path W3492
SFTOF3D
SFTON3D P029
MOVJ C00683 BC00683 VJ=100.00  +MOVJ EC00683 VJ=100.00
SMOVL C00684 BC00684 V=800.0  +MOVJ EC00684
SMOVL C00685 BC00685 V=150.0 PL=0  +MOVJ EC00685
ARCON
SFTON3D P037
SMOVL C00686 BC00686 V=10.0  +MOVJ EC00686
SFTON3D P039
SMOVL C00687 BC00687 V=10.0  +MOVJ EC00687
SMOVL C00688 BC00688 V=10.0  +MOVJ EC00688
ARCOF
SMOVL C00689 BC00689 V=800.0  +MOVJ EC00689
SMOVL C00690 BC00690 V=1000.0  +MOVJ EC00690
SFTOF3D
'EndPath W3492
MOVJ C00691 BC00691 VJ=100.00  +MOVJ EC00691 VJ=100.00
MOVJ C00692 BC00692 VJ=100.00  +MOVJ EC00692 VJ=100.00
'Path W3493
SFTOF3D
SFTON3D P039
MOVJ C00693 BC00693 VJ=100.00  +MOVJ EC00693 VJ=100.00
SMOVL C00694 BC00694 V=800.0  +MOVJ EC00694
SMOVL C00695 BC00695 V=150.0 PL=0  +MOVJ EC00695
ARCON
SFTON3D P040
SMOVL C00696 BC00696 V=10.0  +MOVJ EC00696
SFTON3D P041
SMOVL C00697 BC00697 V=10.0  +MOVJ EC00697
SMOVL C00698 BC00698 V=10.0  +MOVJ EC00698
ARCON
SMOVL C00699 BC00699 V=11.7  +MOVJ EC00699
ARCOF
SMOVL C00700 BC00700 V=800.0  +MOVJ EC00700
SMOVL C00701 BC00701 V=1000.0  +MOVJ EC00701
SFTOF3D
'EndPath W3493
MOVJ C00702 BC00702 VJ=100.00  +MOVJ EC00702 VJ=100.00
MOVJ C00703 BC00703 VJ=100.00  +MOVJ EC00703 VJ=100.00
'16
'Path W3491
SFTOF3D
SFTON3D P080
MOVJ C00704 BC00704 VJ=100.00  +MOVJ EC00704 VJ=100.00
SMOVL C00705 BC00705 V=800.0  +MOVJ EC00705
SMOVL C00706 BC00706 V=150.0 PL=0  +MOVJ EC00706
ARCON
SMOVL C00707 BC00707 V=10.0  +MOVJ EC00707
SFTON3D P044
SMOVL C00708 BC00708 V=10.0  +MOVJ EC00708
SMOVL C00709 BC00709 V=10.0  +MOVJ EC00709
ARCOF
SMOVL C00710 BC00710 V=800.0  +MOVJ EC00710
SMOVL C00711 BC00711 V=1000.0  +MOVJ EC00711
SFTOF3D
'EndPath W3491
MOVJ C00712 BC00712 VJ=100.00  +MOVJ EC00712 VJ=100.00
'Path W3492
SFTOF3D
SFTON3D P080
MOVJ C00713 BC00713 VJ=100.00  +MOVJ EC00713 VJ=100.00
SMOVL C00714 BC00714 V=800.0  +MOVJ EC00714
SMOVL C00715 BC00715 V=150.0 PL=0  +MOVJ EC00715
ARCON
SFTON3D P042
SMOVL C00716 BC00716 V=10.0  +MOVJ EC00716
SFTON3D P043
SMOVL C00717 BC00717 V=10.0  +MOVJ EC00717
SMOVL C00718 BC00718 V=10.0  +MOVJ EC00718
ARCOF
SMOVL C00719 BC00719 V=800.0  +MOVJ EC00719
SMOVL C00720 BC00720 V=1000.0  +MOVJ EC00720
SFTOF3D
'EndPath W3492
MOVJ C00721 BC00721 VJ=100.00  +MOVJ EC00721 VJ=100.00
MOVJ C00722 BC00722 VJ=100.00  +MOVJ EC00722 VJ=100.00
'Path W3493
SFTOF3D
SFTON3D P044
MOVJ C00723 BC00723 VJ=100.00  +MOVJ EC00723 VJ=100.00
SMOVL C00724 BC00724 V=800.0  +MOVJ EC00724
SMOVL C00725 BC00725 V=150.0 PL=0  +MOVJ EC00725
ARCON
SFTON3D P045
SMOVL C00726 BC00726 V=10.0  +MOVJ EC00726
SFTON3D P046
SMOVL C00727 BC00727 V=10.0  +MOVJ EC00727
SMOVL C00728 BC00728 V=10.0  +MOVJ EC00728
ARCOF
SMOVL C00729 BC00729 V=800.0  +MOVJ EC00729
SMOVL C00730 BC00730 V=1000.0  +MOVJ EC00730
SFTOF3D
'EndPath W3493
MOVJ C00731 BC00731 VJ=100.00  +MOVJ EC00731 VJ=100.00
MOVJ C00732 BC00732 VJ=100.00  +MOVJ EC00732 VJ=100.00
'17
'Path W3494
SFTOF3D
SFTON3D P027
MOVJ C00733 BC00733 VJ=100.00  +MOVJ EC00733 VJ=100.00
SMOVL C00734 BC00734 V=800.0  +MOVJ EC00734
SMOVL C00735 BC00735 V=150.0 PL=0  +MOVJ EC00735
ARCON
SMOVL C00736 BC00736 V=10.0  +MOVJ EC00736
ARCOF
SMOVL C00737 BC00737 V=800.0  +MOVJ EC00737
SMOVL C00738 BC00738 V=1000.0  +MOVJ EC00738
SFTOF3D
'EndPath W3494
'Path W3495
SFTOF3D
SFTON3D P027
MOVJ C00739 BC00739 VJ=100.00  +MOVJ EC00739 VJ=100.00
SMOVL C00740 BC00740 V=800.0  +MOVJ EC00740
SMOVL C00741 BC00741 V=150.0 PL=0  +MOVJ EC00741
ARCON
SMOVL C00742 BC00742 V=10.8  +MOVJ EC00742
ARCOF
SMOVL C00743 BC00743 V=800.0  +MOVJ EC00743
SMOVL C00744 BC00744 V=1000.0  +MOVJ EC00744
SFTOF3D
'EndPath W3495
'Path W3496
SFTOF3D
SFTON3D P027
MOVJ C00745 BC00745 VJ=100.00  +MOVJ EC00745 VJ=100.00
SFTOF3D
'EndPath W3496
MOVJ C00746 BC00746 VJ=100.00  +MOVJ EC00746 VJ=100.00
MOVJ C00747 BC00747 VJ=100.00  +MOVJ EC00747 VJ=100.00
MOVJ C00748 BC00748 VJ=100.00  +MOVJ EC00748 VJ=100.00
'18
'Path W3497
SFTOF3D
SFTON3D P024
MOVJ C00749 BC00749 VJ=100.00  +MOVJ EC00749 VJ=100.00
SMOVL C00750 BC00750 V=800.0  +MOVJ EC00750
SMOVL C00751 BC00751 V=150.0 PL=0  +MOVJ EC00751
ARCON
SWVON WEV#(16)
SMOVL C00752 BC00752 V=9.2  +MOVJ EC00752
SFTON3D P036
SMOVL C00753 BC00753 V=9.2  +MOVJ EC00753
SMOVL C00754 BC00754 V=9.2  +MOVJ EC00754
SFTON3D P035
SMOVL C00755 BC00755 V=9.2  +MOVJ EC00755
ARCOF
SWVOF
SMOVL C00756 BC00756 V=800.0  +MOVJ EC00756
SMOVL C00757 BC00757 V=1000.0  +MOVJ EC00757
SFTOF3D
'EndPath W3497
'
'Path W4855
SFTOF3D
SFTON3D P071
MOVJ C00758 BC00758 VJ=100.00  +MOVJ EC00758 VJ=100.00
SMOVL C00759 BC00759 V=800.0  +MOVJ EC00759
MACRO1 MJ#(0) ARGF9
SMOVL C00760 BC00760 V=150.0 PL=0  +MOVJ EC00760
ARCON
SWVON WEV#(16)
SMOVL C00761 BC00761 V=8.8  +MOVJ EC00761
SFTON3D P072
SMOVL C00762 BC00762 V=8.8  +MOVJ EC00762
SMOVL C00763 BC00763 V=8.8  +MOVJ EC00763
ARCOF
SWVOF
SMOVL C00764 BC00764 V=166.7  +MOVJ EC00764
SMOVL C00765 BC00765 V=800.0  +MOVJ EC00765
SFTOF3D
COMM SMOVL C00766 BC00766 V=800.0  +MOVJ EC00766
COMM SMOVL C00767 BC00767 V=800.0  +MOVJ EC00767
COMM SFTON3D P072
COMM SMOVL C00768 BC00768 V=166.7 PL=0  +MOVJ EC00768
COMM ARCON
COMM SMOVL C00769 BC00769 V=8.8  +MOVJ EC00769
COMM SMOVL C00770 BC00770 V=8.8  +MOVJ EC00770
COMM SMOVL C00771 BC00771 V=8.8  +MOVJ EC00771
COMM SMOVL C00772 BC00772 V=8.8  +MOVJ EC00772
COMM ARCOF
COMM MOVL C00773 BC00773 V=166.7  +MOVJ EC00773 VJ=0.78
COMM SMOVL C00774 BC00774 V=1000.0  +MOVJ EC00774
COMM SFTOF3D
COMM 'EndPath W4855
'
'
MOVJ C00775 BC00775 VJ=100.00  +MOVJ EC00775 VJ=100.00
'19
MOVJ C00776 BC00776 VJ=100.00  +MOVJ EC00776 VJ=100.00
'Path W3499
SFTOF3D
SFTON3D P023
MOVJ C00777 BC00777 VJ=100.00  +MOVJ EC00777 VJ=100.00
SMOVL C00778 BC00778 V=800.0  +MOVJ EC00778
SMOVL C00779 BC00779 V=150.0 PL=0  +MOVJ EC00779
MACRO1 MJ#(0) ARGF6
ARCON
SWVON WEV#(66)
SMOVL C00780 BC00780 V=7.5  +MOVJ EC00780
SMOVL C00781 BC00781 V=7.5  +MOVJ EC00781
SMOVL C00782 BC00782 V=7.5  +MOVJ EC00782
ARCOF
SWVOF
SMOVL C00783 BC00783 V=800.0  +MOVJ EC00783
SMOVL C00784 BC00784 V=1000.0  +MOVJ EC00784
SFTOF3D
'EndPath W3499
MOVJ C00785 BC00785 VJ=100.00  +MOVJ EC00785 VJ=100.00
'Path W3500
SFTOF3D
SFTON3D P034
MOVJ C00786 BC00786 VJ=100.00  +MOVJ EC00786 VJ=100.00
SMOVL C00787 BC00787 V=800.0  +MOVJ EC00787
MACRO1 MJ#(0) ARGF9
SMOVL C00788 BC00788 V=150.0 PL=0  +MOVJ EC00788
ARCON
SMOVL C00789 BC00789 V=8.3  +MOVJ EC00789
SFTON3D P050
SMOVL C00790 BC00790 V=8.3  +MOVJ EC00790
SMOVL C00791 BC00791 V=8.3  +MOVJ EC00791
ARCOF
SMOVL C00792 BC00792 V=800.0  +MOVJ EC00792
SMOVL C00793 BC00793 V=1000.0  +MOVJ EC00793
SFTOF3D
'EndPath W3500
'Path W3501
SFTOF3D
SFTON3D P051
MOVJ C00794 BC00794 VJ=100.00  +MOVJ EC00794 VJ=100.00
SMOVL C00795 BC00795 V=800.0  +MOVJ EC00795
SMOVL C00796 BC00796 V=150.0 PL=0  +MOVJ EC00796
ARCON
SMOVL C00797 BC00797 V=7.5  +MOVJ EC00797
SMOVL C00798 BC00798 V=7.5  +MOVJ EC00798
SMOVL C00799 BC00799 V=7.5  +MOVJ EC00799
ARCOF
SWVOF
SMOVL C00800 BC00800 V=800.0  +MOVJ EC00800
SMOVL C00801 BC00801 V=1000.0  +MOVJ EC00801
SFTOF3D
'EndPath W3501
MOVJ C00802 BC00802 VJ=100.00  +MOVJ EC00802 VJ=100.00
'20
MOVJ C00803 BC00803 VJ=100.00  +MOVJ EC00803 VJ=100.00
MOVJ C00804 BC00804 VJ=100.00  +MOVJ EC00804 VJ=100.00
'offset 5mm
'Path W3500
SFTOF3D
SFTON3D P032
MOVJ C00805 BC00805 VJ=100.00  +MOVJ EC00805 VJ=100.00
SMOVL C00806 BC00806 V=800.0  +MOVJ EC00806
SMOVL C00807 BC00807 V=150.0 PL=0  +MOVJ EC00807
ARCON
SMOVL C00808 BC00808 V=9.2  +MOVJ EC00808
ARCOF
SMOVL C00809 BC00809 V=800.0  +MOVJ EC00809
SMOVL C00810 BC00810 V=1000.0  +MOVJ EC00810
SFTOF3D
'EndPath W3500
SFTOF3D
'EndPath W3502
'offset 5mm
'Path W3503
SFTOF3D
SFTON3D P032
MOVJ C00811 BC00811 VJ=100.00  +MOVJ EC00811 VJ=100.00
SMOVL C00812 BC00812 V=800.0  +MOVJ EC00812
SMOVL C00813 BC00813 V=150.0 PL=0  +MOVJ EC00813
ARCON
SMOVL C00814 BC00814 V=10.0  +MOVJ EC00814
ARCOF
SMOVL C00815 BC00815 V=800.0  +MOVJ EC00815
SMOVL C00816 BC00816 V=1000.0  +MOVJ EC00816
SFTOF3D
'EndPath W3503
MOVJ C00817 BC00817 VJ=100.00  +MOVJ EC00817 VJ=100.00
'Path W3504
SFTOF3D
SFTON3D P032
MOVJ C00818 BC00818 VJ=100.00  +MOVJ EC00818 VJ=100.00
SMOVL C00819 BC00819 V=800.0  +MOVJ EC00819
SMOVL C00820 BC00820 V=150.0 PL=0  +MOVJ EC00820
ARCON
SMOVL C00821 BC00821 V=11.7  +MOVJ EC00821
SMOVL C00822 BC00822 V=11.7  +MOVJ EC00822
ARCOF
SMOVL C00823 BC00823 V=800.0  +MOVJ EC00823
SMOVL C00824 BC00824 V=1000.0  +MOVJ EC00824
SFTOF3D
'EndPath W3504
MOVJ C00825 BC00825 VJ=100.00  +MOVJ EC00825 VJ=100.00
'21
MOVJ C00826 BC00826 VJ=100.00  +MOVJ EC00826 VJ=100.00
'Path W3505
SFTOF3D
SFTON3D P097
MOVJ C00827 BC00827 VJ=100.00  +MOVJ EC00827 VJ=100.00
SMOVL C00828 BC00828 V=800.0  +MOVJ EC00828
SMOVL C00829 BC00829 V=150.0 PL=0  +MOVJ EC00829
ARCON
SMOVL C00830 BC00830 V=10.8  +MOVJ EC00830
SFTON3D P021
SMOVL C00831 BC00831 V=10.8  +MOVJ EC00831
SFTON3D P022
SMOVL C00832 BC00832 V=10.8  +MOVJ EC00832
SMOVL C00833 BC00833 V=11.7  +MOVJ EC00833
ARCOF
SMOVL C00834 BC00834 V=800.0  +MOVJ EC00834
SMOVL C00835 BC00835 V=1000.0  +MOVJ EC00835
SFTOF3D
'EndPath W3505
MOVJ C00836 BC00836 VJ=100.00  +MOVJ EC00836 VJ=100.00
'Path W3506
SFTOF3D
SFTON3D P095
MOVJ C00837 BC00837 VJ=100.00  +MOVJ EC00837 VJ=100.00
SMOVL C00838 BC00838 V=800.0  +MOVJ EC00838
SMOVL C00839 BC00839 V=150.0 PL=0  +MOVJ EC00839
MACRO1 MJ#(0) ARGF14
ARCON
SMOVL C00840 BC00840 V=10.0  +MOVJ EC00840
SMOVL C00841 BC00841 V=10.0  +MOVJ EC00841
SMOVL C00842 BC00842 V=10.0  +MOVJ EC00842
ARCOF
SMOVL C00843 BC00843 V=800.0  +MOVJ EC00843
SMOVL C00844 BC00844 V=1000.0  +MOVJ EC00844
SFTOF3D
'EndPath W3506
'Path W3507
SFTOF3D
SFTON3D P096
MOVJ C00845 BC00845 VJ=100.00  +MOVJ EC00845 VJ=100.00
SMOVL C00846 BC00846 V=800.0  +MOVJ EC00846
SMOVL C00847 BC00847 V=150.0 PL=0  +MOVJ EC00847
ARCON
SMOVL C00848 BC00848 V=10.0  +MOVJ EC00848
SMOVL C00849 BC00849 V=10.0  +MOVJ EC00849
ARCOF
SMOVL C00850 BC00850 V=800.0  +MOVJ EC00850
SMOVL C00851 BC00851 V=1000.0  +MOVJ EC00851
SFTOF3D
'EndPath W3507
MOVJ C00852 BC00852 VJ=100.00  +MOVJ EC00852 VJ=100.00
MOVJ C00853 BC00853 VJ=100.00  +MOVJ EC00853 VJ=100.00
'Path W4856
SFTOF3D
SFTON3D P071
MOVJ C00854 BC00854 VJ=100.00  +MOVJ EC00854 VJ=100.00
SMOVL C00855 BC00855 V=800.0  +MOVJ EC00855
SMOVL C00856 BC00856 V=150.0 PL=0  +MOVJ EC00856
ARCON
SMOVL C00857 BC00857 V=8.3  +MOVJ EC00857
SFTON3D P073
SMOVL C00858 BC00858 V=8.3  +MOVJ EC00858
SMOVL C00859 BC00859 V=8.3  +MOVJ EC00859
ARCOF
SMOVL C00860 BC00860 V=800.0  +MOVJ EC00860
SMOVL C00861 BC00861 V=1000.0  +MOVJ EC00861
SFTOF3D
'EndPath W4856
MOVJ C00862 BC00862 VJ=100.00  +MOVJ EC00862 VJ=100.00
MOVJ C00863 BC00863 VJ=50.00  +MOVJ EC00863 VJ=0.78
MOVJ C00864 BC00864 VJ=100.00  +MOVJ EC00864 VJ=50.00
COMM SFTON3D P080
COMM SMOVL C00865 BC00865 V=800.0  +MOVJ EC00865
COMM SMOVL C00866 BC00866 V=150.0 PL=0  +MOVJ EC00866
COMM ARCON
COMM SMOVL C00867 BC00867 V=8.3  +MOVJ EC00867
COMM SMOVL C00868 BC00868 V=8.3  +MOVJ EC00868
COMM SMOVC C00869 BC00869 V=8.3  +MOVJ EC00869
COMM ARCOF
COMM SMOVL C00870 BC00870 V=800.0  +MOVJ EC00870
SFTOF3D
SMOVL C00871 BC00871 V=1000.0  +MOVJ EC00871
MOVJ C00872 BC00872 VJ=100.00  +MOVJ EC00872 VJ=100.00
MOVJ C00873 BC00873 VJ=100.00  +MOVJ EC00873 VJ=100.00
MOVJ C00874 BC00874 VJ=100.00  +MOVJ EC00874 VJ=100.00
MOVJ C00875 BC00875 VJ=100.00  +MOVJ EC00875 VJ=100.00
SFTON3D P081
SMOVL C00876 BC00876 V=666.7  +MOVJ EC00876
SMOVL C00877 BC00877 V=166.7 PL=0  +MOVJ EC00877
ARCON
SMOVL C00878 BC00878 V=8.3  +MOVJ EC00878
SFTON3D P074
SMOVL C00879 BC00879 V=8.3  +MOVJ EC00879
SMOVL C00880 BC00880 V=8.3  +MOVJ EC00880
ARCOF
SMOVL C00881 BC00881 V=333.3  +MOVJ EC00881
SFTOF3D
MOVL C00882 BC00882 V=1000.0  +MOVJ EC00882 VJ=100.00
MOVJ C00883 BC00883 VJ=100.00  +MOVJ EC00883 VJ=100.00
MOVJ C00884 BC00884 VJ=100.00  +MOVJ EC00884 VJ=100.00
'cut_wire_dol
'cut_wire_dol
'cut_wire_dol
CALL JOB:CLEAN-R1_KM_3P
COMM 'X2_8A-21A(90,0)
COMM MOVJ C00885 BC00885 VJ=100.00  +MOVJ EC00885 VJ=100.00
COMM CALL JOB:CLEAN-R1_KM_NEW
COMM MOVJ C00886 BC00886 VJ=100.00  +MOVJ EC00886 VJ=100.00
COMM MOVJ C00887 BC00887 VJ=100.00  +MOVJ EC00887 VJ=100.00
COMM 'Path S3463
COMM SFTOF3D
COMM MOVJ C00888 BC00888 VJ=100.00  +MOVJ EC00888 VJ=100.00
COMM MOVL C00889 BC00889 V=666.7  +MOVJ EC00889 VJ=100.00
COMM SMOVL C00890 BC00890 V=166.7  +MOVJ EC00890
COMM SREFP 3 C00891 BC00891  +REFP EC00891
COMM CALL JOB:SEARCH-R1-S13D
COMM SET P095 P006
COMM SFTON3D P095
COMM SMOVL C00892 BC00892 V=166.7  +MOVJ EC00892
COMM SMOVL C00893 BC00893 V=166.7  +MOVJ EC00893
COMM SREFP 3 C00894 BC00894  +REFP EC00894
COMM CALL JOB:SEARCH-R1-S13D
COMM SET P095 P006
COMM SFTON3D P095
COMM SMOVL C00895 BC00895 V=166.7  +MOVJ EC00895
COMM MOVL C00896 BC00896 V=1000.0  +MOVJ EC00896 VJ=100.00
COMM 'EndPath S3463
COMM 'Path S3464
COMM SFTOF3D
COMM MOVJ C00897 BC00897 VJ=100.00  +MOVJ EC00897 VJ=100.00
COMM MOVL C00898 BC00898 V=666.7  +MOVJ EC00898 VJ=100.00
COMM SMOVL C00899 BC00899 V=166.7  +MOVJ EC00899
COMM SREFP 3 C00900 BC00900  +REFP EC00900
COMM CALL JOB:SEARCH-R1-S13D
COMM SET P096 P006
COMM SFTON3D P096
COMM SMOVL C00901 BC00901 V=166.7  +MOVJ EC00901
COMM SREFP 3 C00902 BC00902  +REFP EC00902
COMM CALL JOB:SEARCH-R1-S13D
COMM SET P096 P006
COMM SFTON3D P096
COMM SMOVL C00903 BC00903 V=166.7  +MOVJ EC00903
COMM MOVL C00904 BC00904 V=1000.0  +MOVJ EC00904 VJ=100.00
COMM 'EndPath S3464
COMM 'Path S3465
COMM SFTOF3D
COMM MOVJ C00905 BC00905 VJ=100.00  +MOVJ EC00905 VJ=100.00
COMM MOVL C00906 BC00906 V=666.7  +MOVJ EC00906 VJ=100.00
COMM SMOVL C00907 BC00907 V=166.7  +MOVJ EC00907
COMM SREFP 3 C00908 BC00908  +REFP EC00908
COMM CALL JOB:SEARCH-R1-S13D
COMM SET P021 P006
COMM SFTON3D P021
COMM SMOVL C00909 BC00909 V=166.7  +MOVJ EC00909
COMM SMOVL C00910 BC00910 V=166.7  +MOVJ EC00910
COMM SREFP 3 C00911 BC00911  +REFP EC00911
COMM CALL JOB:SEARCH-R1-S13D
COMM SET P021 P006
COMM SFTON3D P021
COMM SMOVL C00912 BC00912 V=166.7  +MOVJ EC00912
COMM MOVL C00913 BC00913 V=1000.0  +MOVJ EC00913 VJ=100.00
COMM 'EndPath S3465
COMM 'Path S3464
COMM SFTOF3D
COMM MOVJ C00914 BC00914 VJ=100.00  +MOVJ EC00914 VJ=100.00
COMM MOVL C00915 BC00915 V=666.7  +MOVJ EC00915 VJ=100.00
COMM SMOVL C00916 BC00916 V=166.7  +MOVJ EC00916
COMM SREFP 3 C00917 BC00917  +REFP EC00917
COMM CALL JOB:SEARCH-R1-S13D
COMM SET P022 P006
COMM SFTON3D P022
COMM SMOVL C00918 BC00918 V=166.7  +MOVJ EC00918
COMM SREFP 3 C00919 BC00919  +REFP EC00919
COMM CALL JOB:SEARCH-R1-S13D
COMM SET P022 P006
COMM SFTON3D P022
COMM SMOVL C00920 BC00920 V=166.7  +MOVJ EC00920
COMM MOVL C00921 BC00921 V=1000.0  +MOVJ EC00921 VJ=100.00
COMM 'EndPath S3464
COMM MOVJ C00922 BC00922 VJ=100.00  +MOVJ EC00922 VJ=100.00
COMM 'Path S3465
COMM SFTOF3D
COMM MOVJ C00923 BC00923 VJ=100.00  +MOVJ EC00923 VJ=100.00
COMM MOVL C00924 BC00924 V=666.7  +MOVJ EC00924 VJ=100.00
COMM SMOVL C00925 BC00925 V=166.7  +MOVJ EC00925
COMM SREFP 3 C00926 BC00926  +REFP EC00926
COMM CALL JOB:SEARCH-R1-S13D
COMM SET P050 P006
COMM SFTON3D P050
COMM SMOVL C00927 BC00927 V=166.7  +MOVJ EC00927
COMM SREFP 3 C00928 BC00928  +REFP EC00928
COMM CALL JOB:SEARCH-R1-S13D
COMM SET P050 P006
COMM SFTON3D P050
COMM SMOVL C00929 BC00929 V=166.7  +MOVJ EC00929
COMM SMOVL C00930 BC00930 V=166.7  +MOVJ EC00930
COMM SREFP 3 C00931 BC00931  +REFP EC00931
COMM CALL JOB:SEARCH-R1-S13D
COMM SET P050 P006
COMM SFTON3D P050
COMM SMOVL C00932 BC00932 V=166.7  +MOVJ EC00932
COMM MOVL C00933 BC00933 V=1000.0  +MOVJ EC00933 VJ=100.00
COMM 'EndPath S3465
COMM 'Path S3466
COMM SFTOF3D
COMM MOVJ C00934 BC00934 VJ=100.00  +MOVJ EC00934 VJ=100.00
COMM MOVL C00935 BC00935 V=666.7  +MOVJ EC00935 VJ=100.00
COMM SMOVL C00936 BC00936 V=166.7  +MOVJ EC00936
COMM SREFP 3 C00937 BC00937  +REFP EC00937
COMM CALL JOB:SEARCH-R1-S13D
COMM SET P051 P006
COMM SFTON3D P051
COMM SMOVL C00938 BC00938 V=166.7  +MOVJ EC00938
COMM SREFP 3 C00939 BC00939  +REFP EC00939
COMM CALL JOB:SEARCH-R1-S13D
COMM SET P051 P006
COMM SFTON3D P051
COMM SMOVL C00940 BC00940 V=166.7  +MOVJ EC00940
COMM SMOVL C00941 BC00941 V=250.0  +MOVJ EC00941
COMM SREFP 3 C00942 BC00942  +REFP EC00942
COMM CALL JOB:SEARCH-R1-S13D
COMM SET P051 P006
COMM SFTON3D P051
COMM SMOVL C00943 BC00943 V=166.7  +MOVJ EC00943
COMM MOVL C00944 BC00944 V=1000.0  +MOVJ EC00944 VJ=100.00
COMM 'EndPath S3466
COMM MOVJ C00945 BC00945 VJ=100.00  +MOVJ EC00945 VJ=100.00
COMM MOVJ C00946 BC00946 VJ=100.00  +MOVJ EC00946 VJ=100.00
COMM 'Path S3467
COMM SFTOF3D
COMM MOVJ C00947 BC00947 VJ=100.00  +MOVJ EC00947 VJ=100.00
COMM MOVL C00948 BC00948 V=666.7  +MOVJ EC00948 VJ=100.00
COMM SMOVL C00949 BC00949 V=166.7  +MOVJ EC00949
COMM SREFP 3 C00950 BC00950  +REFP EC00950
COMM CALL JOB:SEARCH-R1-S13D
COMM SET P054 P006
COMM SFTON3D P054
COMM SMOVL C00951 BC00951 V=250.0  +MOVJ EC00951
COMM SMOVL C00952 BC00952 V=166.7  +MOVJ EC00952
COMM SREFP 3 C00953 BC00953  +REFP EC00953
COMM CALL JOB:SEARCH-R1-S13D
COMM SET P054 P006
COMM SFTON3D P054
COMM SMOVL C00954 BC00954 V=166.7  +MOVJ EC00954
COMM SMOVL C00955 BC00955 V=800.0  +MOVJ EC00955
COMM SMOVL C00956 BC00956 V=166.7  +MOVJ EC00956
COMM SREFP 3 C00957 BC00957  +REFP EC00957
COMM CALL JOB:SEARCH-R1-S13D
COMM SET P054 P006
COMM SFTON3D P054
COMM SMOVL C00958 BC00958 V=166.7  +MOVJ EC00958
COMM MOVL C00959 BC00959 V=1000.0  +MOVJ EC00959 VJ=100.00
COMM 'EndPath S3467
COMM 'Path S3475
COMM SFTOF3D
COMM MOVJ C00960 BC00960 VJ=100.00  +MOVJ EC00960 VJ=100.00
COMM MOVL C00961 BC00961 V=666.7  +MOVJ EC00961 VJ=100.00
COMM SMOVL C00962 BC00962 V=166.7  +MOVJ EC00962
COMM SREFP 3 C00963 BC00963  +REFP EC00963
COMM CALL JOB:SEARCH-R1-S13D
COMM SET P034 P006
COMM SFTON3D P034
COMM SMOVL C00964 BC00964 V=166.7  +MOVJ EC00964
COMM SMOVL C00965 BC00965 V=333.3  +MOVJ EC00965
COMM SMOVL C00966 BC00966 V=166.7  +MOVJ EC00966
COMM SREFP 3 C00967 BC00967  +REFP EC00967
COMM CALL JOB:SEARCH-R1-S13D
COMM SET P034 P006
COMM SFTON3D P034
COMM SMOVL C00968 BC00968 V=166.7  +MOVJ EC00968
COMM SMOVL C00969 BC00969 V=166.7  +MOVJ EC00969
COMM SREFP 3 C00970 BC00970  +REFP EC00970
COMM CALL JOB:SEARCH-R1-S13D
COMM SET P034 P006
COMM SFTON3D P034
COMM SMOVL C00971 BC00971 V=166.7  +MOVJ EC00971
COMM MOVL C00972 BC00972 V=1000.0  +MOVJ EC00972 VJ=100.00
COMM 'EndPath S3475
COMM 'Path S3464
COMM SFTOF3D
COMM MOVJ C00973 BC00973 VJ=100.00  +MOVJ EC00973 VJ=100.00
COMM MOVL C00974 BC00974 V=666.7  +MOVJ EC00974 VJ=100.00
COMM SMOVL C00975 BC00975 V=166.7  +MOVJ EC00975
COMM SREFP 3 C00976 BC00976  +REFP EC00976
COMM CALL JOB:SEARCH-R1-S13D
COMM SET P023 P006
COMM SFTON3D P023
COMM SMOVL C00977 BC00977 V=166.7  +MOVJ EC00977
COMM SMOVL C00978 BC00978 V=500.0  +MOVJ EC00978
COMM SMOVL C00979 BC00979 V=166.7  +MOVJ EC00979
COMM SREFP 3 C00980 BC00980  +REFP EC00980
COMM CALL JOB:SEARCH-R1-S13D
COMM SET P023 P006
COMM SFTON3D P023
COMM SMOVL C00981 BC00981 V=166.7  +MOVJ EC00981
COMM SMOVL C00982 BC00982 V=166.7  +MOVJ EC00982
COMM SREFP 3 C00983 BC00983  +REFP EC00983
COMM CALL JOB:SEARCH-R1-S13D
COMM SET P023 P006
COMM SFTON3D P023
COMM SMOVL C00984 BC00984 V=166.7  +MOVJ EC00984
COMM MOVL C00985 BC00985 V=1000.0  +MOVJ EC00985 VJ=100.00
COMM MOVJ C00986 BC00986 VJ=80.00  +MOVJ EC00986 VJ=80.00
COMM MOVJ C00987 BC00987 VJ=80.00  +MOVJ EC00987 VJ=80.00
COMM SFTOF3D
COMM MOVJ C00988 BC00988 VJ=80.00  +MOVJ EC00988 VJ=80.00
COMM SMOVL C00989 BC00989 V=166.7  +MOVJ EC00989
COMM SREFP 3 C00990 BC00990  +REFP EC00990
COMM CALL JOB:SEARCH-R1-S13D
COMM SET P061 P006
COMM SFTON3D P061
COMM SMOVL C00991 BC00991 V=166.7  +MOVJ EC00991
COMM SREFP 3 C00992 BC00992  +REFP EC00992
COMM CALL JOB:SEARCH-R1-S13D
COMM SET P061 P006
COMM SFTON3D P061
COMM SMOVL C00993 BC00993 V=166.7  +MOVJ EC00993
COMM SFTOF3D
COMM SMOVL C00994 BC00994 V=500.0  +MOVJ EC00994
COMM SMOVL C00995 BC00995 V=166.7  +MOVJ EC00995
COMM SREFP 3 C00996 BC00996  +REFP EC00996
COMM CALL JOB:SEARCH-R1-S13D
COMM SET P062 P006
COMM SFTON3D P062
COMM SMOVL C00997 BC00997 V=166.7  +MOVJ EC00997
COMM SREFP 3 C00998 BC00998  +REFP EC00998
COMM CALL JOB:SEARCH-R1-S13D
COMM SET P062 P006
COMM SFTON3D P062
COMM SMOVL C00999 BC00999 V=166.7  +MOVJ EC00999
COMM SFTOF3D
COMM SMOVL C01000 BC01000 V=500.0  +MOVJ EC01000
COMM SMOVL C01001 BC01001 V=166.7  +MOVJ EC01001
COMM SREFP 3 C01002 BC01002  +REFP EC01002
COMM CALL JOB:SEARCH-R1-S13D
COMM SET P063 P006
COMM SFTON3D P063
COMM SMOVL C01003 BC01003 V=166.7  +MOVJ EC01003
COMM SREFP 3 C01004 BC01004  +REFP EC01004
COMM CALL JOB:SEARCH-R1-S13D
COMM SET P063 P006
COMM SFTON3D P063
COMM SMOVL C01005 BC01005 V=166.7  +MOVJ EC01005
COMM SFTOF3D
COMM SMOVL C01006 BC01006 V=500.0  +MOVJ EC01006
COMM MOVJ C01007 BC01007 VJ=80.00  +MOVJ EC01007 VJ=80.00
COMM MOVJ C01008 BC01008 VJ=80.00  +MOVJ EC01008 VJ=80.00
COMM 'EndPath S3464
COMM MOVJ C01009 BC01009 VJ=100.00  +MOVJ EC01009 VJ=100.00
COMM 'Path S3465
COMM SFTOF3D
COMM MOVJ C01010 BC01010 VJ=100.00  +MOVJ EC01010 VJ=100.00
COMM MOVL C01011 BC01011 V=666.7  +MOVJ EC01011 VJ=100.00
COMM SMOVL C01012 BC01012 V=166.7  +MOVJ EC01012
COMM SREFP 3 C01013 BC01013  +REFP EC01013
COMM CALL JOB:SEARCH-R1-S13D
COMM SET P024 P006
COMM SFTON3D P024
COMM SMOVL C01014 BC01014 V=166.7  +MOVJ EC01014
COMM SREFP 3 C01015 BC01015  +REFP EC01015
COMM CALL JOB:SEARCH-R1-S13D
COMM SET P024 P006
COMM SFTON3D P024
COMM SMOVL C01016 BC01016 V=166.7  +MOVJ EC01016
COMM SMOVL C01017 BC01017 V=166.7  +MOVJ EC01017
COMM SREFP 3 C01018 BC01018  +REFP EC01018
COMM CALL JOB:SEARCH-R1-S13D
COMM SET P024 P006
COMM SFTON3D P024
COMM SMOVL C01019 BC01019 V=166.7  +MOVJ EC01019
COMM MOVL C01020 BC01020 V=1000.0  +MOVJ EC01020 VJ=100.00
COMM 'EndPath S3465
COMM 'Path S3476
COMM SFTOF3D
COMM MOVJ C01021 BC01021 VJ=100.00  +MOVJ EC01021 VJ=100.00
COMM MOVL C01022 BC01022 V=666.7  +MOVJ EC01022 VJ=100.00
COMM SMOVL C01023 BC01023 V=166.7  +MOVJ EC01023
COMM SREFP 3 C01024 BC01024  +REFP EC01024
COMM CALL JOB:SEARCH-R1-S13D
COMM SET P035 P006
COMM SFTON3D P035
COMM SMOVL C01025 BC01025 V=166.7  +MOVJ EC01025
COMM SREFP 3 C01026 BC01026  +REFP EC01026
COMM CALL JOB:SEARCH-R1-S13D
COMM SET P035 P006
COMM SFTON3D P035
COMM SMOVL C01027 BC01027 V=166.7  +MOVJ EC01027
COMM SMOVL C01028 BC01028 V=333.3  +MOVJ EC01028
COMM SMOVL C01029 BC01029 V=166.7  +MOVJ EC01029
COMM SREFP 3 C01030 BC01030  +REFP EC01030
COMM CALL JOB:SEARCH-R1-S13D
COMM SET P035 P006
COMM SFTON3D P035
COMM SMOVL C01031 BC01031 V=166.7  +MOVJ EC01031
COMM MOVL C01032 BC01032 V=1000.0  +MOVJ EC01032 VJ=100.00
COMM 'EndPath S3476
COMM 'Path S3470
COMM SFTOF3D
COMM MOVJ C01033 BC01033 VJ=100.00  +MOVJ EC01033 VJ=100.00
COMM MOVL C01034 BC01034 V=666.7  +MOVJ EC01034 VJ=100.00
COMM SMOVL C01035 BC01035 V=166.7  +MOVJ EC01035
COMM SREFP 3 C01036 BC01036  +REFP EC01036
COMM CALL JOB:SEARCH-R1-S13D
COMM SET P029 P006
COMM SFTON3D P029
COMM SMOVL C01037 BC01037 V=166.7  +MOVJ EC01037
COMM SREFP 3 C01038 BC01038  +REFP EC01038
COMM CALL JOB:SEARCH-R1-S13D
COMM SET P029 P006
COMM SFTON3D P029
COMM SMOVL C01039 BC01039 V=166.7  +MOVJ EC01039
COMM SMOVL C01040 BC01040 V=250.0  +MOVJ EC01040
COMM SMOVL C01041 BC01041 V=166.7  +MOVJ EC01041
COMM SREFP 3 C01042 BC01042  +REFP EC01042
COMM CALL JOB:SEARCH-R1-S13D
COMM SET P029 P006
COMM SFTON3D P029
COMM SMOVL C01043 BC01043 V=166.7  +MOVJ EC01043
COMM MOVL C01044 BC01044 V=1000.0  +MOVJ EC01044 VJ=100.00
COMM 'EndPath S3470
COMM 'Path S4850
COMM SFTOF3D
COMM MOVL C01045 BC01045 V=666.7  +MOVJ EC01045 VJ=100.00
COMM SMOVL C01046 BC01046 V=166.7  +MOVJ EC01046
COMM SREFP 3 C01047 BC01047  +REFP EC01047
COMM CALL JOB:SEARCH-R1-S13D
COMM SET P071 P006
COMM SFTON3D P071
COMM SMOVL C01048 BC01048 V=166.7  +MOVJ EC01048
COMM SREFP 3 C01049 BC01049  +REFP EC01049
COMM CALL JOB:SEARCH-R1-S13D
COMM SET P071 P006
COMM SFTON3D P071
COMM SMOVL C01050 BC01050 V=166.7  +MOVJ EC01050
COMM SMOVL C01051 BC01051 V=166.7  +MOVJ EC01051
COMM SREFP 3 C01052 BC01052  +REFP EC01052
COMM CALL JOB:SEARCH-R1-S13D
COMM SET P071 P006
COMM SFTON3D P071
COMM SMOVL C01053 BC01053 V=166.7  +MOVJ EC01053
COMM MOVL C01054 BC01054 V=1000.0  +MOVJ EC01054 VJ=100.00
COMM 'EndPath S4850
COMM 'Path S4851
COMM SFTOF3D
COMM MOVJ C01055 BC01055 VJ=100.00  +MOVJ EC01055 VJ=100.00
COMM 'POMIAR_DOD_WZM_BOK
COMM MOVL C01056 BC01056 V=666.7  +MOVJ EC01056 VJ=100.00
COMM SMOVL C01057 BC01057 V=166.7  +MOVJ EC01057
COMM SREFP 3 C01058 BC01058  +REFP EC01058
COMM CALL JOB:SEARCH-R1-S13D
COMM SET P080 P006
COMM SFTON3D P080
COMM SMOVL C01059 BC01059 V=166.7  +MOVJ EC01059
COMM SREFP 3 C01060 BC01060  +REFP EC01060
COMM CALL JOB:SEARCH-R1-S13D
COMM SET P080 P006
COMM SFTON3D P080
COMM SMOVL C01061 BC01061 V=166.7  +MOVJ EC01061
COMM SMOVL C01062 BC01062 V=250.0  +MOVJ EC01062
COMM SMOVL C01063 BC01063 V=166.7  +MOVJ EC01063
COMM SREFP 3 C01064 BC01064  +REFP EC01064
COMM CALL JOB:SEARCH-R1-S13D
COMM SET P080 P006
COMM SFTON3D P080
COMM SMOVL C01065 BC01065 V=166.7  +MOVJ EC01065
COMM MOVL C01066 BC01066 V=1000.0  +MOVJ EC01066 VJ=100.00
COMM SFTOF3D
COMM MOVJ C01067 BC01067 VJ=100.00  +MOVJ EC01067 VJ=100.00
COMM MOVL C01068 BC01068 V=666.7  +MOVJ EC01068 VJ=100.00
COMM SMOVL C01069 BC01069 V=166.7  +MOVJ EC01069
COMM SREFP 3 C01070 BC01070  +REFP EC01070
COMM CALL JOB:SEARCH-R1-S13D
COMM SET P072 P006
COMM SFTON3D P072
COMM SMOVL C01071 BC01071 V=166.7  +MOVJ EC01071
COMM SREFP 3 C01072 BC01072  +REFP EC01072
COMM CALL JOB:SEARCH-R1-S13D
COMM SET P072 P006
COMM SFTON3D P072
COMM SMOVL C01073 BC01073 V=166.7  +MOVJ EC01073
COMM MOVL C01074 BC01074 V=1000.0  +MOVJ EC01074 VJ=100.00
COMM 'EndPath S4851
COMM MOVJ C01075 BC01075 VJ=100.00  +MOVJ EC01075 VJ=100.00
COMM MOVJ C01076 BC01076 VJ=100.00  +MOVJ EC01076 VJ=100.00
COMM 'Path S4852
COMM SFTOF3D
COMM MOVJ C01077 BC01077 VJ=100.00  +MOVJ EC01077 VJ=100.00
COMM MOVL C01078 BC01078 V=666.7  +MOVJ EC01078 VJ=100.00
COMM SMOVL C01079 BC01079 V=166.7  +MOVJ EC01079
COMM SREFP 3 C01080 BC01080  +REFP EC01080
COMM CALL JOB:SEARCH-R1-S13D
COMM SET P073 P006
COMM SFTON3D P073
COMM SMOVL C01081 BC01081 V=166.7  +MOVJ EC01081
COMM SMOVL C01082 BC01082 V=166.7  +MOVJ EC01082
COMM SREFP 3 C01083 BC01083  +REFP EC01083
COMM CALL JOB:SEARCH-R1-S13D
COMM SET P073 P006
COMM SFTON3D P073
COMM SMOVL C01084 BC01084 V=166.7  +MOVJ EC01084
COMM SMOVL C01085 BC01085 V=166.7  +MOVJ EC01085
COMM SREFP 3 C01086 BC01086  +REFP EC01086
COMM CALL JOB:SEARCH-R1-S13D
COMM SET P073 P006
COMM SFTON3D P073
COMM SMOVL C01087 BC01087 V=166.7  +MOVJ EC01087
COMM MOVL C01088 BC01088 V=1000.0  +MOVJ EC01088 VJ=100.00
COMM 'EndPath S4852
COMM MOVJ C01089 BC01089 VJ=100.00  +MOVJ EC01089 VJ=100.00
COMM 'Path S4853
COMM SFTOF3D
COMM MOVJ C01090 BC01090 VJ=100.00  +MOVJ EC01090 VJ=100.00
COMM MOVL C01091 BC01091 V=666.7  +MOVJ EC01091 VJ=100.00
COMM SMOVL C01092 BC01092 V=166.7  +MOVJ EC01092
COMM SREFP 3 C01093 BC01093  +REFP EC01093
COMM CALL JOB:SEARCH-R1-S13D
COMM SET P074 P006
COMM SFTON3D P074
COMM SMOVL C01094 BC01094 V=166.7  +MOVJ EC01094
COMM SREFP 3 C01095 BC01095  +REFP EC01095
COMM CALL JOB:SEARCH-R1-S13D
COMM SET P074 P006
COMM SFTON3D P074
COMM SMOVL C01096 BC01096 V=166.7  +MOVJ EC01096
COMM MOVL C01097 BC01097 V=1000.0  +MOVJ EC01097 VJ=100.00
COMM 'EndPath S4853
COMM 'Path S3467
COMM SFTOF3D
COMM MOVJ C01098 BC01098 VJ=100.00  +MOVJ EC01098 VJ=100.00
COMM MOVJ C01099 BC01099 VJ=100.00  +MOVJ EC01099 VJ=100.00
COMM MOVL C01100 BC01100 V=666.7  +MOVJ EC01100 VJ=100.00
COMM SMOVL C01101 BC01101 V=166.7  +MOVJ EC01101
COMM SREFP 3 C01102 BC01102  +REFP EC01102
COMM CALL JOB:SEARCH-R1-S13D
COMM SET P081 P006
COMM SFTON3D P081
COMM SMOVL C01103 BC01103 V=166.7  +MOVJ EC01103
COMM SMOVL C01104 BC01104 V=166.7  +MOVJ EC01104
COMM SREFP 3 C01105 BC01105  +REFP EC01105
COMM CALL JOB:SEARCH-R1-S13D
COMM SET P081 P006
COMM SFTON3D P081
COMM SMOVL C01106 BC01106 V=166.7  +MOVJ EC01106
COMM SMOVL C01107 BC01107 V=800.0  +MOVJ EC01107
COMM SMOVL C01108 BC01108 V=166.7  +MOVJ EC01108
COMM SREFP 3 C01109 BC01109  +REFP EC01109
COMM CALL JOB:SEARCH-R1-S13D
COMM SET P081 P006
COMM SFTON3D P081
COMM SMOVL C01110 BC01110 V=166.7  +MOVJ EC01110
COMM MOVJ C01111 BC01111 VJ=100.00  +MOVJ EC01111 VJ=100.00
COMM MOVJ C01112 BC01112 VJ=100.00  +MOVJ EC01112 VJ=100.00
COMM SFTOF3D
COMM MOVJ C01113 BC01113 VJ=100.00  +MOVJ EC01113 VJ=100.00
COMM MOVL C01114 BC01114 V=666.7  +MOVJ EC01114 VJ=100.00
COMM SMOVL C01115 BC01115 V=166.7  +MOVJ EC01115
COMM SREFP 3 C01116 BC01116  +REFP EC01116
COMM CALL JOB:SEARCH-R1-S13D
COMM SET P026 P006
COMM SFTON3D P026
COMM SMOVL C01117 BC01117 V=166.7  +MOVJ EC01117
COMM SREFP 3 C01118 BC01118  +REFP EC01118
COMM CALL JOB:SEARCH-R1-S13D
COMM SET P026 P006
COMM SFTON3D P026
COMM SMOVL C01119 BC01119 V=166.7  +MOVJ EC01119
COMM SMOVL C01120 BC01120 V=800.0  +MOVJ EC01120
COMM SMOVL C01121 BC01121 V=166.7  +MOVJ EC01121
COMM SREFP 3 C01122 BC01122  +REFP EC01122
COMM CALL JOB:SEARCH-R1-S13D
COMM SET P026 P006
COMM SFTON3D P026
COMM SMOVL C01123 BC01123 V=166.7  +MOVJ EC01123
COMM MOVL C01124 BC01124 V=1000.0  +MOVJ EC01124 VJ=100.00
COMM 'EndPath S3467
COMM MOVJ C01125 BC01125 VJ=100.00  +MOVJ EC01125 VJ=100.00
COMM 'Path S3466
COMM SFTOF3D
COMM MOVJ C01126 BC01126 VJ=100.00  +MOVJ EC01126 VJ=100.00
COMM MOVL C01127 BC01127 V=666.7  +MOVJ EC01127 VJ=100.00
COMM SMOVL C01128 BC01128 V=166.7  +MOVJ EC01128
COMM SREFP 3 C01129 BC01129  +REFP EC01129
COMM CALL JOB:SEARCH-R1-S13D
COMM SET P025 P006
COMM SFTON3D P025
COMM SMOVL C01130 BC01130 V=166.7  +MOVJ EC01130
COMM SMOVL C01131 BC01131 V=166.7  +MOVJ EC01131
COMM SREFP 3 C01132 BC01132  +REFP EC01132
COMM CALL JOB:SEARCH-R1-S13D
COMM SET P025 P006
COMM SFTON3D P025
COMM SMOVL C01133 BC01133 V=166.7  +MOVJ EC01133
COMM SMOVL C01134 BC01134 V=200.0  +MOVJ EC01134
COMM SMOVL C01135 BC01135 V=166.7  +MOVJ EC01135
COMM SREFP 3 C01136 BC01136  +REFP EC01136
COMM CALL JOB:SEARCH-R1-S13D
COMM SET P025 P006
COMM SFTON3D P025
COMM SMOVL C01137 BC01137 V=166.7  +MOVJ EC01137
COMM MOVL C01138 BC01138 V=1000.0  +MOVJ EC01138 VJ=100.00
COMM 'EndPath S3466
COMM MOVJ C01139 BC01139 VJ=100.00  +MOVJ EC01139 VJ=100.00
COMM 'Path S3469
COMM SFTOF3D
COMM MOVJ C01140 BC01140 VJ=100.00  +MOVJ EC01140 VJ=100.00
COMM MOVL C01141 BC01141 V=666.7  +MOVJ EC01141 VJ=100.00
COMM SMOVL C01142 BC01142 V=166.7  +MOVJ EC01142
COMM SREFP 3 C01143 BC01143  +REFP EC01143
COMM CALL JOB:SEARCH-R1-S13D
COMM SET P028 P006
COMM SFTON3D P028
COMM SMOVL C01144 BC01144 V=166.7  +MOVJ EC01144
COMM SREFP 3 C01145 BC01145  +REFP EC01145
COMM CALL JOB:SEARCH-R1-S13D
COMM SET P028 P006
COMM SFTON3D P028
COMM SMOVL C01146 BC01146 V=166.7  +MOVJ EC01146
COMM SMOVL C01147 BC01147 V=333.3  +MOVJ EC01147
COMM SMOVL C01148 BC01148 V=166.7  +MOVJ EC01148
COMM SREFP 3 C01149 BC01149  +REFP EC01149
COMM CALL JOB:SEARCH-R1-S13D
COMM SET P028 P006
COMM SFTON3D P028
COMM SMOVL C01150 BC01150 V=166.7  +MOVJ EC01150
COMM MOVL C01151 BC01151 V=1000.0  +MOVJ EC01151 VJ=100.00
COMM 'EndPath S3469
COMM MOVJ C01152 BC01152 VJ=100.00  +MOVJ EC01152 VJ=100.00
COMM 'Path S3474
COMM SFTOF3D
COMM MOVJ C01153 BC01153 VJ=100.00  +MOVJ EC01153 VJ=100.00
COMM MOVL C01154 BC01154 V=666.7  +MOVJ EC01154 VJ=100.00
COMM SMOVL C01155 BC01155 V=166.7  +MOVJ EC01155
COMM SREFP 3 C01156 BC01156  +REFP EC01156
COMM CALL JOB:SEARCH-R1-S13D
COMM SET P033 P006
COMM SFTON3D P033
COMM SMOVL C01157 BC01157 V=166.7  +MOVJ EC01157
COMM SREFP 3 C01158 BC01158  +REFP EC01158
COMM CALL JOB:SEARCH-R1-S13D
COMM SET P033 P006
COMM SFTON3D P033
COMM SMOVL C01159 BC01159 V=166.7  +MOVJ EC01159
COMM SMOVL C01160 BC01160 V=250.0  +MOVJ EC01160
COMM SMOVL C01161 BC01161 V=166.7  +MOVJ EC01161
COMM SREFP 3 C01162 BC01162  +REFP EC01162
COMM CALL JOB:SEARCH-R1-S13D
COMM SET P033 P006
COMM SFTON3D P033
COMM SMOVL C01163 BC01163 V=166.7  +MOVJ EC01163
COMM MOVL C01164 BC01164 V=1000.0  +MOVJ EC01164 VJ=100.00
COMM 'EndPath S3474
COMM 'Path S3468
COMM SFTOF3D
COMM MOVJ C01165 BC01165 VJ=100.00  +MOVJ EC01165 VJ=100.00
COMM MOVL C01166 BC01166 V=666.7  +MOVJ EC01166 VJ=100.00
COMM SMOVL C01167 BC01167 V=166.7  +MOVJ EC01167
COMM SREFP 3 C01168 BC01168  +REFP EC01168
COMM CALL JOB:SEARCH-R1-S13D
COMM SET P027 P006
COMM SFTON3D P027
COMM SMOVL C01169 BC01169 V=166.7  +MOVJ EC01169
COMM SMOVL C01170 BC01170 V=166.7  +MOVJ EC01170
COMM SREFP 3 C01171 BC01171  +REFP EC01171
COMM CALL JOB:SEARCH-R1-S13D
COMM SET P027 P006
COMM SFTON3D P027
COMM SMOVL C01172 BC01172 V=166.7  +MOVJ EC01172
COMM SMOVL C01173 BC01173 V=166.7  +MOVJ EC01173
COMM SREFP 3 C01174 BC01174  +REFP EC01174
COMM CALL JOB:SEARCH-R1-S13D
COMM SET P027 P006
COMM SFTON3D P027
COMM SMOVL C01175 BC01175 V=166.7  +MOVJ EC01175
COMM MOVL C01176 BC01176 V=1000.0  +MOVJ EC01176 VJ=100.00
COMM 'EndPath S3468
COMM 'Path S3471
COMM SFTOF3D
COMM MOVJ C01177 BC01177 VJ=100.00  +MOVJ EC01177 VJ=100.00
COMM MOVL C01178 BC01178 V=666.7  +MOVJ EC01178 VJ=100.00
COMM SMOVL C01179 BC01179 V=166.7  +MOVJ EC01179
COMM SREFP 3 C01180 BC01180  +REFP EC01180
COMM CALL JOB:SEARCH-R1-S13D
COMM SET P030 P006
COMM SFTON3D P030
COMM SMOVL C01181 BC01181 V=166.7  +MOVJ EC01181
COMM SREFP 3 C01182 BC01182  +REFP EC01182
COMM CALL JOB:SEARCH-R1-S13D
COMM SET P030 P006
COMM SFTON3D P030
COMM SMOVL C01183 BC01183 V=166.7  +MOVJ EC01183
COMM MOVL C01184 BC01184 V=1000.0  +MOVJ EC01184 VJ=100.00
COMM 'EndPath S3471
COMM 'Path S3472
COMM SFTOF3D
COMM MOVJ C01185 BC01185 VJ=100.00  +MOVJ EC01185 VJ=100.00
COMM MOVL C01186 BC01186 V=666.7  +MOVJ EC01186 VJ=100.00
COMM SMOVL C01187 BC01187 V=166.7  +MOVJ EC01187
COMM SREFP 3 C01188 BC01188  +REFP EC01188
COMM CALL JOB:SEARCH-R1-S13D
COMM SET P031 P006
COMM SFTON3D P031
COMM SMOVL C01189 BC01189 V=166.7  +MOVJ EC01189
COMM SREFP 3 C01190 BC01190  +REFP EC01190
COMM CALL JOB:SEARCH-R1-S13D
COMM SET P031 P006
COMM SFTON3D P031
COMM SMOVL C01191 BC01191 V=166.7  +MOVJ EC01191
COMM MOVL C01192 BC01192 V=1000.0  +MOVJ EC01192 VJ=100.00
COMM 'EndPath S3472
COMM MOVJ C01193 BC01193 VJ=100.00  +MOVJ EC01193 VJ=100.00
COMM 'Path S3472
COMM SFTOF3D
COMM MOVJ C01194 BC01194 VJ=100.00  +MOVJ EC01194 VJ=100.00
COMM MOVL C01195 BC01195 V=666.7  +MOVJ EC01195 VJ=100.00
COMM SMOVL C01196 BC01196 V=166.7  +MOVJ EC01196
COMM SREFP 3 C01197 BC01197  +REFP EC01197
COMM CALL JOB:SEARCH-R1-S13D
COMM SET P032 P006
COMM SFTON3D P032
COMM SMOVL C01198 BC01198 V=166.7  +MOVJ EC01198
COMM SREFP 3 C01199 BC01199  +REFP EC01199
COMM CALL JOB:SEARCH-R1-S13D
COMM SET P032 P006
COMM SFTON3D P032
COMM SMOVL C01200 BC01200 V=166.7  +MOVJ EC01200
COMM SMOVL C01201 BC01201 V=133.3  +MOVJ EC01201
COMM SREFP 3 C01202 BC01202  +REFP EC01202
COMM CALL JOB:SEARCH-R1-S13D
COMM SET P032 P006
COMM SFTON3D P032
COMM SMOVL C01203 BC01203 V=166.7  +MOVJ EC01203
COMM MOVL C01204 BC01204 V=1000.0  +MOVJ EC01204 VJ=100.00
COMM 'EndPath S3472
COMM MOVJ C01205 BC01205 VJ=100.00  +MOVJ EC01205 VJ=100.00
COMM 'Path S3477
COMM SFTOF3D
COMM MOVJ C01206 BC01206 VJ=100.00  +MOVJ EC01206 VJ=100.00
COMM SMOVL C01207 BC01207 V=166.7  +MOVJ EC01207
COMM SREFP 3 C01208 BC01208  +REFP EC01208
COMM CALL JOB:SEARCH-R1-S13D
COMM SET P069 P006
COMM SFTON3D P069
COMM SMOVL C01209 BC01209 V=250.0  +MOVJ EC01209
COMM SMOVL C01210 BC01210 V=250.0  +MOVJ EC01210
COMM SMOVL C01211 BC01211 V=166.7  +MOVJ EC01211
COMM SREFP 3 C01212 BC01212  +REFP EC01212
COMM CALL JOB:SEARCH-R1-S13D
COMM SET P069 P006
COMM SFTON3D P069
COMM SMOVL C01213 BC01213 V=166.7  +MOVJ EC01213
COMM SFTOF3D
COMM SMOVL C01214 BC01214 V=666.7  +MOVJ EC01214
COMM MOVL C01215 BC01215 V=666.7  +MOVJ EC01215 VJ=100.00
COMM SMOVL C01216 BC01216 V=166.7  +MOVJ EC01216
COMM SREFP 3 C01217 BC01217  +REFP EC01217
COMM CALL JOB:SEARCH-R1-S13D
COMM SET P052 P006
COMM SFTON3D P052
COMM SMOVL C01218 BC01218 V=166.7  +MOVJ EC01218
COMM SREFP 3 C01219 BC01219  +REFP EC01219
COMM CALL JOB:SEARCH-R1-S13D
COMM SET P052 P006
COMM SFTON3D P052
COMM SMOVL C01220 BC01220 V=166.7  +MOVJ EC01220
COMM MOVL C01221 BC01221 V=1000.0  +MOVJ EC01221 VJ=100.00
COMM 'EndPath S3477
COMM MOVJ C01222 BC01222 VJ=100.00  +MOVJ EC01222 VJ=100.00
COMM 'poprawi searcha- nie mialem
COMM 'wyciecia
COMM 'Path S3478
COMM SFTOF3D
COMM MOVJ C01223 BC01223 VJ=100.00  +MOVJ EC01223 VJ=100.00
COMM MOVL C01224 BC01224 V=666.7  +MOVJ EC01224 VJ=100.00
COMM SMOVL C01225 BC01225 V=166.7  +MOVJ EC01225
COMM SREFP 3 C01226 BC01226  +REFP EC01226
COMM CALL JOB:SEARCH-R1-S13D
COMM SET P053 P006
COMM SFTON3D P053
COMM SMOVL C01227 BC01227 V=166.7  +MOVJ EC01227
COMM SREFP 3 C01228 BC01228  +REFP EC01228
COMM CALL JOB:SEARCH-R1-S13D
COMM SET P053 P006
COMM SFTON3D P053
COMM SMOVL C01229 BC01229 V=166.7  +MOVJ EC01229
COMM MOVL C01230 BC01230 V=1000.0  +MOVJ EC01230 VJ=100.00
COMM 'EndPath S3478
COMM '
COMM MOVJ C01231 BC01231 VJ=100.00  +MOVJ EC01231 VJ=100.00
COMM 'Path W3476
COMM SFTOF3D
COMM SFTON3D P033
COMM MOVJ C01232 BC01232 VJ=100.00  +MOVJ EC01232 VJ=100.00
COMM SMOVL C01233 BC01233 V=800.0  +MOVJ EC01233
COMM SMOVL C01234 BC01234 V=166.7 PL=0  +MOVJ EC01234
COMM MACRO1 MJ#(0) ARGF14
COMM ARCON
COMM SMOVL C01235 BC01235 V=10.0  +MOVJ EC01235
COMM ARCOF
COMM SMOVL C01236 BC01236 V=800.0  +MOVJ EC01236
COMM SMOVL C01237 BC01237 V=1000.0  +MOVJ EC01237
COMM SFTOF3D
COMM 'EndPath W3476
COMM 'Path W3477
COMM SFTOF3D
COMM SFTON3D P033
COMM MOVJ C01238 BC01238 VJ=100.00  +MOVJ EC01238 VJ=100.00
COMM SMOVL C01239 BC01239 V=800.0  +MOVJ EC01239
COMM SMOVL C01240 BC01240 V=166.7 PL=0  +MOVJ EC01240
COMM SMOVL C01241 BC01241 V=10.0  +MOVJ EC01241
COMM SMOVL C01242 BC01242 V=10.0  +MOVJ EC01242
COMM SMOVL C01243 BC01243 V=10.0  +MOVJ EC01243
COMM ARCOF
COMM SMOVL C01244 BC01244 V=800.0  +MOVJ EC01244
COMM SMOVL C01245 BC01245 V=1000.0  +MOVJ EC01245
COMM SFTOF3D
COMM 'EndPath W3477
COMM MOVJ C01246 BC01246 VJ=100.00  +MOVJ EC01246 VJ=100.00
COMM 'Path W3478
COMM SFTOF3D
COMM SFTON3D P033
COMM MOVJ C01247 BC01247 VJ=100.00  +MOVJ EC01247 VJ=100.00
COMM SMOVL C01248 BC01248 V=800.0  +MOVJ EC01248
COMM SMOVL C01249 BC01249 V=166.7 PL=0  +MOVJ EC01249
COMM ARCON
COMM SMOVL C01250 BC01250 V=10.0  +MOVJ EC01250
COMM SMOVL C01251 BC01251 V=10.0  +MOVJ EC01251
COMM SMOVL C01252 BC01252 V=10.0  +MOVJ EC01252
COMM ARCOF
COMM SMOVL C01253 BC01253 V=800.0  +MOVJ EC01253
COMM SMOVL C01254 BC01254 V=1000.0  +MOVJ EC01254
COMM SFTOF3D
COMM 'EndPath W3478
COMM MOVJ C01255 BC01255 VJ=100.00  +MOVJ EC01255 VJ=100.00
COMM MOVJ C01256 BC01256 VJ=100.00  +MOVJ EC01256 VJ=100.00
COMM SFTOF3D
COMM SFTON3D P081
COMM MOVJ C01257 BC01257 VJ=100.00  +MOVJ EC01257 VJ=100.00
COMM SMOVL C01258 BC01258 V=800.0  +MOVJ EC01258
COMM SMOVL C01259 BC01259 V=166.7 PL=0  +MOVJ EC01259
COMM ARCON
COMM SMOVL C01260 BC01260 V=9.2  +MOVJ EC01260
COMM ARCOF
COMM SMOVL C01261 BC01261 V=800.0  +MOVJ EC01261
COMM SMOVL C01262 BC01262 V=1000.0  +MOVJ EC01262
COMM SFTOF3D
COMM 'EndPath W3479
COMM 'Path W3480
COMM SFTOF3D
COMM SFTON3D P081
COMM MOVJ C01263 BC01263 VJ=100.00  +MOVJ EC01263 VJ=100.00
COMM SMOVL C01264 BC01264 V=800.0  +MOVJ EC01264
COMM SMOVL C01265 BC01265 V=150.0 PL=0  +MOVJ EC01265
COMM ARCON
COMM SMOVL C01266 BC01266 V=10.0  +MOVJ EC01266
COMM ARCOF
COMM SMOVL C01267 BC01267 V=800.0  +MOVJ EC01267
COMM SMOVL C01268 BC01268 V=1000.0  +MOVJ EC01268
COMM SFTOF3D
COMM 'EndPath W3480
COMM 'Path W3481
COMM SFTOF3D
COMM SFTON3D P081
COMM MOVJ C01269 BC01269 VJ=100.00  +MOVJ EC01269 VJ=100.00
COMM SMOVL C01270 BC01270 V=800.0  +MOVJ EC01270
COMM SMOVL C01271 BC01271 V=150.0 PL=0  +MOVJ EC01271
COMM ARCON
COMM SMOVL C01272 BC01272 V=10.0  +MOVJ EC01272
COMM ARCOF
COMM SMOVL C01273 BC01273 V=800.0  +MOVJ EC01273
COMM SMOVL C01274 BC01274 V=1000.0  +MOVJ EC01274
COMM SFTOF3D
COMM 'EndPath W3481
COMM MOVJ C01275 BC01275 VJ=100.00  +MOVJ EC01275 VJ=100.00
COMM 'uwaga na podajnik
COMM 'Path W3481
COMM SFTOF3D
COMM SFTON3D P081
COMM MOVJ C01276 BC01276 VJ=50.00  +MOVJ EC01276 VJ=15.00
COMM SMOVL C01277 BC01277 V=800.0  +MOVJ EC01277
COMM SMOVL C01278 BC01278 V=150.0 PL=0  +MOVJ EC01278
COMM ARCON
COMM SMOVL C01279 BC01279 V=10.0  +MOVJ EC01279
COMM ARCOF
COMM SMOVL C01280 BC01280 V=800.0  +MOVJ EC01280
COMM SMOVL C01281 BC01281 V=1000.0  +MOVJ EC01281
COMM SFTOF3D
COMM '9
COMM 'Path W3479
COMM MOVJ C01282 BC01282 VJ=100.00  +MOVJ EC01282 VJ=100.00
COMM SFTOF3D
COMM SFTON3D P026
COMM MOVJ C01283 BC01283 VJ=100.00  +MOVJ EC01283 VJ=100.00
COMM SMOVL C01284 BC01284 V=800.0  +MOVJ EC01284
COMM SMOVL C01285 BC01285 V=166.7 PL=0  +MOVJ EC01285
COMM ARCON
COMM SMOVL C01286 BC01286 V=9.2  +MOVJ EC01286
COMM SMOVL C01287 BC01287 V=9.2  +MOVJ EC01287
COMM SMOVL C01288 BC01288 V=9.2  +MOVJ EC01288
COMM ARCOF
COMM SMOVL C01289 BC01289 V=800.0  +MOVJ EC01289
COMM SMOVL C01290 BC01290 V=1000.0  +MOVJ EC01290
COMM SFTOF3D
COMM 'EndPath W3479
COMM 'Path W3480
COMM SFTOF3D
COMM SFTON3D P026
COMM MOVJ C01291 BC01291 VJ=100.00  +MOVJ EC01291 VJ=100.00
COMM SMOVL C01292 BC01292 V=800.0  +MOVJ EC01292
COMM SMOVL C01293 BC01293 V=150.0 PL=0  +MOVJ EC01293
COMM ARCON
COMM SMOVL C01294 BC01294 V=10.0  +MOVJ EC01294
COMM SMOVL C01295 BC01295 V=10.0  +MOVJ EC01295
COMM SMOVL C01296 BC01296 V=10.0  +MOVJ EC01296
COMM ARCOF
COMM SMOVL C01297 BC01297 V=800.0  +MOVJ EC01297
COMM SMOVL C01298 BC01298 V=1000.0  +MOVJ EC01298
COMM SFTOF3D
COMM 'EndPath W3480
COMM 'Path W3481
COMM SFTOF3D
COMM SFTON3D P026
COMM MOVJ C01299 BC01299 VJ=100.00  +MOVJ EC01299 VJ=100.00
COMM SMOVL C01300 BC01300 V=800.0  +MOVJ EC01300
COMM SMOVL C01301 BC01301 V=150.0 PL=0  +MOVJ EC01301
COMM ARCON
COMM SMOVL C01302 BC01302 V=10.0  +MOVJ EC01302
COMM ARCOF
COMM SMOVL C01303 BC01303 V=800.0  +MOVJ EC01303
COMM SMOVL C01304 BC01304 V=1000.0  +MOVJ EC01304
COMM SFTOF3D
COMM 'EndPath W3481
COMM MOVJ C01305 BC01305 VJ=100.00  +MOVJ EC01305 VJ=100.00
COMM 'uwaga na podajnik
COMM 'Path W3481
COMM SFTOF3D
COMM SFTON3D P026
COMM MOVJ C01306 BC01306 VJ=50.00  +MOVJ EC01306 VJ=15.00
COMM SMOVL C01307 BC01307 V=800.0  +MOVJ EC01307
COMM SMOVL C01308 BC01308 V=150.0 PL=0  +MOVJ EC01308
COMM ARCON
COMM SMOVL C01309 BC01309 V=10.0  +MOVJ EC01309
COMM SMOVL C01310 BC01310 V=10.0  +MOVJ EC01310
COMM ARCOF
COMM SMOVL C01311 BC01311 V=800.0  +MOVJ EC01311
COMM SMOVL C01312 BC01312 V=1000.0  +MOVJ EC01312
COMM SFTOF3D
COMM 'EndPath W3481
COMM 'brak dostepu offset drutu 1cm
COMM 'Path W3482
COMM SFTOF3D
COMM SFTON3D P026
COMM MOVJ C01313 BC01313 VJ=100.00  +MOVJ EC01313 VJ=100.00
COMM SMOVL C01314 BC01314 V=800.0  +MOVJ EC01314
COMM SMOVL C01315 BC01315 V=150.0 PL=0  +MOVJ EC01315
COMM ARCON
COMM SMOVL C01316 BC01316 V=10.0  +MOVJ EC01316
COMM ARCOF
COMM SMOVL C01317 BC01317 V=800.0  +MOVJ EC01317
COMM SMOVL C01318 BC01318 V=1000.0  +MOVJ EC01318
COMM SFTOF3D
COMM 'EndPath W3482
COMM MOVJ C01319 BC01319 VJ=100.00  +MOVJ EC01319 VJ=100.00
COMM MOVJ C01320 BC01320 VJ=100.00  +MOVJ EC01320 VJ=100.00
COMM '10
COMM '11
COMM 'Path W3484
COMM SFTOF3D
COMM SFTON3D P025
COMM MOVJ C01321 BC01321 VJ=100.00  +MOVJ EC01321 VJ=100.00
COMM SMOVL C01322 BC01322 V=800.0  +MOVJ EC01322
COMM SMOVL C01323 BC01323 V=150.0 PL=0  +MOVJ EC01323
COMM ARCON
COMM SMOVL C01324 BC01324 V=10.0  +MOVJ EC01324
COMM SMOVL C01325 BC01325 V=10.0  +MOVJ EC01325
COMM ARCOF
COMM SMOVL C01326 BC01326 V=800.0  +MOVJ EC01326
COMM SMOVL C01327 BC01327 V=1000.0  +MOVJ EC01327
COMM SFTOF3D
COMM 'EndPath W3484
COMM MOVJ C01328 BC01328 VJ=100.00  +MOVJ EC01328 VJ=100.00
COMM 'brak dostepu offset drutu 1cm
COMM 'Path W3483
COMM SFTOF3D
COMM SFTON3D P025
COMM MOVJ C01329 BC01329 VJ=100.00  +MOVJ EC01329 VJ=100.00
COMM SMOVL C01330 BC01330 V=800.0  +MOVJ EC01330
COMM SMOVL C01331 BC01331 V=166.7 PL=0  +MOVJ EC01331
COMM ARCON
COMM SMOVL C01332 BC01332 V=10.0  +MOVJ EC01332
COMM ARCOF
COMM SMOVL C01333 BC01333 V=800.0  +MOVJ EC01333
COMM SMOVL C01334 BC01334 V=1000.0  +MOVJ EC01334
COMM SFTOF3D
COMM 'EndPath W3483
COMM MOVJ C01335 BC01335 VJ=100.00  +MOVJ EC01335 VJ=100.00
COMM MOVJ C01336 BC01336 VJ=100.00  +MOVJ EC01336 VJ=100.00
COMM MOVJ C01337 BC01337 VJ=100.00  +MOVJ EC01337 VJ=100.00
COMM 'Path W4854
COMM SFTOF3D
COMM SFTON3D P073
COMM MOVJ C01338 BC01338 VJ=100.00  +MOVJ EC01338 VJ=100.00
COMM SMOVL C01339 BC01339 V=800.0  +MOVJ EC01339
COMM SMOVL C01340 BC01340 V=150.0 PL=0  +MOVJ EC01340
COMM MACRO1 MJ#(0) ARGF9
COMM ARCON
COMM SMOVL C01341 BC01341 V=9.2  +MOVJ EC01341
COMM SFTON3D P074
COMM SMOVL C01342 BC01342 V=9.2  +MOVJ EC01342
COMM SMOVL C01343 BC01343 V=9.2  +MOVJ EC01343
COMM ARCOF
COMM SMOVL C01344 BC01344 V=800.0  +MOVJ EC01344
COMM MOVJ C01345 BC01345 VJ=50.00  +MOVJ EC01345 VJ=100.00
COMM SMOVL C01346 BC01346 V=166.7  +MOVJ EC01346
COMM SMOVL C01347 BC01347 V=166.7  +MOVJ EC01347
COMM SMOVL C01348 BC01348 V=50.0 PL=0  +MOVJ EC01348
COMM ARCON
COMM SMOVL C01349 BC01349 V=9.2  +MOVJ EC01349
COMM SMOVL C01350 BC01350 V=9.2  +MOVJ EC01350
COMM ARCOF
COMM SMOVL C01351 BC01351 V=1000.0  +MOVJ EC01351
COMM SFTOF3D
COMM 'EndPath W4854
COMM '12
COMM MOVJ C01352 BC01352 VJ=100.00  +MOVJ EC01352 VJ=100.00
COMM MOVJ C01353 BC01353 VJ=100.00  +MOVJ EC01353 VJ=100.00
COMM MOVJ C01354 BC01354 VJ=100.00  +MOVJ EC01354 VJ=100.00
COMM 'Path W3485
COMM SFTOF3D
COMM SFTON3D P034
COMM MOVJ C01355 BC01355 VJ=100.00  +MOVJ EC01355 VJ=100.00
COMM SMOVL C01356 BC01356 V=800.0  +MOVJ EC01356
COMM SMOVL C01357 BC01357 V=150.0 PL=0  +MOVJ EC01357
COMM MACRO1 MJ#(0) ARGF14
COMM ARCON
COMM SMOVL C01358 BC01358 V=10.0  +MOVJ EC01358
COMM SMOVL C01359 BC01359 V=10.0  +MOVJ EC01359
COMM SMOVL C01360 BC01360 V=10.0  +MOVJ EC01360
COMM ARCOF
COMM SMOVL C01361 BC01361 V=800.0  +MOVJ EC01361
COMM SMOVL C01362 BC01362 V=1000.0  +MOVJ EC01362
COMM SFTOF3D
COMM MOVJ C01363 BC01363 VJ=80.00  +MOVJ EC01363 VJ=80.00
COMM MOVJ C01364 BC01364 VJ=80.00  +MOVJ EC01364 VJ=80.00
COMM MOVJ C01365 BC01365 VJ=80.00  +MOVJ EC01365 VJ=80.00
COMM MACRO1 MJ#(0) ARGF6
COMM SFTON3D P063
COMM SMOVL C01366 BC01366 V=166.7  +MOVJ EC01366
COMM ARCON
COMM SMOVL C01367 BC01367 V=11.7  +MOVJ EC01367
COMM SMOVL C01368 BC01368 V=11.7  +MOVJ EC01368
COMM SFTON3D P062
COMM SMOVL C01369 BC01369 V=11.0  +MOVJ EC01369
COMM SMOVL C01370 BC01370 V=11.0  +MOVJ EC01370
COMM SFTON3D P061
COMM SMOVL C01371 BC01371 V=11.0  +MOVJ EC01371
COMM SMOVL C01372 BC01372 V=11.0  +MOVJ EC01372
COMM ARCOF
COMM SMOVL C01373 BC01373 V=800.0  +MOVJ EC01373
COMM SFTOF3D
COMM MOVJ C01374 BC01374 VJ=80.00  +MOVJ EC01374 VJ=80.00
COMM MOVJ C01375 BC01375 VJ=80.00  +MOVJ EC01375 VJ=80.00
COMM MOVJ C01376 BC01376 VJ=80.00  +MOVJ EC01376 VJ=80.00
COMM 'EndPath W3485
COMM 'Path W3486
COMM SFTOF3D
COMM SFTON3D P050
COMM MOVJ C01377 BC01377 VJ=100.00  +MOVJ EC01377 VJ=100.00
COMM SMOVL C01378 BC01378 V=800.0  +MOVJ EC01378
COMM SMOVL C01379 BC01379 V=150.0 PL=0  +MOVJ EC01379
COMM MACRO1 MJ#(0) ARGF14
COMM ARCON
COMM SMOVL C01380 BC01380 V=10.0  +MOVJ EC01380
COMM SMOVL C01381 BC01381 V=10.0  +MOVJ EC01381
COMM SMOVL C01382 BC01382 V=10.0  +MOVJ EC01382
COMM ARCOF
COMM SMOVL C01383 BC01383 V=800.0  +MOVJ EC01383
COMM SMOVL C01384 BC01384 V=1000.0  +MOVJ EC01384
COMM SFTOF3D
COMM 'EndPath W3486
COMM MOVJ C01385 BC01385 VJ=100.00  +MOVJ EC01385 VJ=100.00
COMM 'Path W3485
COMM SFTOF3D
COMM SFTON3D P034
COMM MOVJ C01386 BC01386 VJ=100.00  +MOVJ EC01386 VJ=100.00
COMM SMOVL C01387 BC01387 V=800.0  +MOVJ EC01387
COMM SMOVL C01388 BC01388 V=166.7 PL=0  +MOVJ EC01388
COMM ARCON
COMM SMOVL C01389 BC01389 V=9.2  +MOVJ EC01389
COMM SMOVL C01390 BC01390 V=9.2  +MOVJ EC01390
COMM SMOVL C01391 BC01391 V=9.2  +MOVJ EC01391
COMM ARCOF
COMM SMOVL C01392 BC01392 V=800.0  +MOVJ EC01392
COMM SMOVL C01393 BC01393 V=1000.0  +MOVJ EC01393
COMM SFTOF3D
COMM 'EndPath W3485
COMM 'Path W3487
COMM SFTOF3D
COMM SFTON3D P054
COMM MOVJ C01394 BC01394 VJ=100.00  +MOVJ EC01394 VJ=100.00
COMM SMOVL C01395 BC01395 V=800.0  +MOVJ EC01395
COMM SMOVL C01396 BC01396 V=150.0 PL=0  +MOVJ EC01396
COMM ARCON
COMM SMOVL C01397 BC01397 V=9.2  +MOVJ EC01397
COMM SMOVL C01398 BC01398 V=9.2  +MOVJ EC01398
COMM SMOVL C01399 BC01399 V=9.2  +MOVJ EC01399
COMM ARCOF
COMM SMOVL C01400 BC01400 V=800.0  +MOVJ EC01400
COMM SMOVL C01401 BC01401 V=1000.0  +MOVJ EC01401
COMM SFTOF3D
COMM 'EndPath W3487
COMM MOVJ C01402 BC01402 VJ=100.00  +MOVJ EC01402 VJ=100.00
COMM 'Path W3487
COMM SFTOF3D
COMM SFTON3D P028
COMM MOVJ C01403 BC01403 VJ=100.00  +MOVJ EC01403 VJ=100.00
COMM SMOVL C01404 BC01404 V=800.0  +MOVJ EC01404
COMM SMOVL C01405 BC01405 V=150.0 PL=0  +MOVJ EC01405
COMM ARCON
COMM SMOVL C01406 BC01406 V=9.2  +MOVJ EC01406
COMM SMOVL C01407 BC01407 V=9.2  +MOVJ EC01407
COMM SMOVL C01408 BC01408 V=9.2  +MOVJ EC01408
COMM ARCOF
COMM SMOVL C01409 BC01409 V=800.0  +MOVJ EC01409
COMM SMOVL C01410 BC01410 V=1000.0  +MOVJ EC01410
COMM SFTOF3D
COMM 'EndPath W3487
COMM MOVJ C01411 BC01411 VJ=100.00  +MOVJ EC01411 VJ=100.00
COMM MOVJ C01412 BC01412 VJ=100.00  +MOVJ EC01412 VJ=100.00
COMM 'brak dostepu offset 5mm
COMM 'Path W3488
COMM SFTOF3D
COMM SFTON3D P028
COMM MOVJ C01413 BC01413 VJ=100.00  +MOVJ EC01413 VJ=100.00
COMM SMOVL C01414 BC01414 V=800.0  +MOVJ EC01414
COMM SMOVL C01415 BC01415 V=150.0 PL=0  +MOVJ EC01415
COMM ARCON
COMM SMOVL C01416 BC01416 V=11.7  +MOVJ EC01416
COMM ARCOF
COMM SMOVL C01417 BC01417 V=800.0  +MOVJ EC01417
COMM SMOVL C01418 BC01418 V=1000.0  +MOVJ EC01418
COMM SFTOF3D
COMM 'EndPath W3488
COMM MOVJ C01419 BC01419 VJ=100.00  +MOVJ EC01419 VJ=100.00
COMM '13
COMM 'Path W3489
COMM SFTOF3D
COMM SFTON3D P030
COMM MOVJ C01420 BC01420 VJ=100.00  +MOVJ EC01420 VJ=100.00
COMM SMOVL C01421 BC01421 V=800.0  +MOVJ EC01421
COMM SMOVL C01422 BC01422 V=150.0 PL=0  +MOVJ EC01422
COMM MACRO1 MJ#(0) ARGF9
COMM ARCON
COMM SWVON WEV#(10)
COMM SFTON3D P031
COMM SMOVL C01423 BC01423 V=12.5  +MOVJ EC01423
COMM ARCOF
COMM SWVOF
COMM SMOVL C01424 BC01424 V=800.0  +MOVJ EC01424
COMM SMOVL C01425 BC01425 V=1000.0  +MOVJ EC01425
COMM SFTOF3D
COMM 'EndPath W3489
COMM 'Path W3490
COMM SFTOF3D
COMM MOVJ C01426 BC01426 VJ=100.00  +MOVJ EC01426 VJ=100.00
COMM MACRO1 MJ#(0) ARGF6
COMM SFTON3D P069
COMM SMOVL C01427 BC01427 V=250.0  +MOVJ EC01427
COMM ARCON
COMM SMOVL C01428 BC01428 V=11.7  +MOVJ EC01428
COMM ARCOF
COMM SMOVL C01429 BC01429 V=250.0  +MOVJ EC01429
COMM SFTOF3D
COMM SFTON3D P052
COMM MOVJ C01430 BC01430 VJ=100.00  +MOVJ EC01430 VJ=100.00
COMM SMOVL C01431 BC01431 V=800.0  +MOVJ EC01431
COMM SMOVL C01432 BC01432 V=150.0 PL=0  +MOVJ EC01432
COMM MACRO1 MJ#(0) ARGF14
COMM ARCON
COMM SMOVL C01433 BC01433 V=10.0  +MOVJ EC01433
COMM SMOVL C01434 BC01434 V=10.0  +MOVJ EC01434
COMM SMOVL C01435 BC01435 V=10.0  +MOVJ EC01435
COMM ARCOF
COMM SMOVL C01436 BC01436 V=800.0  +MOVJ EC01436
COMM SMOVL C01437 BC01437 V=1000.0  +MOVJ EC01437
COMM SFTOF3D
COMM 'EndPath W3490
COMM MOVJ C01438 BC01438 VJ=100.00  +MOVJ EC01438 VJ=100.00
COMM 'poprawic spoine - nie mialem w
COMM 'yciecia
COMM 'Path W3491
COMM SFTOF3D
COMM SFTON3D P053
COMM MOVJ C01439 BC01439 VJ=100.00  +MOVJ EC01439 VJ=100.00
COMM SMOVL C01440 BC01440 V=800.0  +MOVJ EC01440
COMM SMOVL C01441 BC01441 V=150.0 PL=0  +MOVJ EC01441
COMM ARCON
COMM SMOVL C01442 BC01442 V=10.0  +MOVJ EC01442
COMM SMOVL C01443 BC01443 V=10.0  +MOVJ EC01443
COMM SMOVL C01444 BC01444 V=10.0  +MOVJ EC01444
COMM ARCOF
COMM SMOVL C01445 BC01445 V=800.0  +MOVJ EC01445
COMM SMOVL C01446 BC01446 V=1000.0  +MOVJ EC01446
COMM SFTOF3D
COMM 'EndPath W3491
COMM '14
COMM '15-brak
COMM MOVJ C01447 BC01447 VJ=100.00  +MOVJ EC01447 VJ=100.00
COMM '16
COMM 'Path W3491
COMM SFTOF3D
COMM SFTON3D P029
COMM MOVJ C01448 BC01448 VJ=100.00  +MOVJ EC01448 VJ=100.00
COMM SMOVL C01449 BC01449 V=800.0  +MOVJ EC01449
COMM SMOVL C01450 BC01450 V=150.0 PL=0  +MOVJ EC01450
COMM ARCON
COMM SMOVL C01451 BC01451 V=10.0  +MOVJ EC01451
COMM SMOVL C01452 BC01452 V=10.0  +MOVJ EC01452
COMM ARCOF
COMM SMOVL C01453 BC01453 V=800.0  +MOVJ EC01453
COMM SMOVL C01454 BC01454 V=1000.0  +MOVJ EC01454
COMM SFTOF3D
COMM 'EndPath W3491
COMM MOVJ C01455 BC01455 VJ=100.00  +MOVJ EC01455 VJ=100.00
COMM 'Path W3492
COMM SFTOF3D
COMM SFTON3D P029
COMM MOVJ C01456 BC01456 VJ=100.00  +MOVJ EC01456 VJ=100.00
COMM SMOVL C01457 BC01457 V=800.0  +MOVJ EC01457
COMM SMOVL C01458 BC01458 V=150.0 PL=0  +MOVJ EC01458
COMM ARCON
COMM SMOVL C01459 BC01459 V=10.0  +MOVJ EC01459
COMM ARCOF
COMM SMOVL C01460 BC01460 V=800.0  +MOVJ EC01460
COMM SMOVL C01461 BC01461 V=1000.0  +MOVJ EC01461
COMM SFTOF3D
COMM 'EndPath W3492
COMM MOVJ C01462 BC01462 VJ=100.00  +MOVJ EC01462 VJ=100.00
COMM MOVJ C01463 BC01463 VJ=100.00  +MOVJ EC01463 VJ=100.00
COMM 'Path W3493
COMM SFTOF3D
COMM SFTON3D P029
COMM MOVJ C01464 BC01464 VJ=100.00  +MOVJ EC01464 VJ=100.00
COMM SMOVL C01465 BC01465 V=800.0  +MOVJ EC01465
COMM SMOVL C01466 BC01466 V=150.0 PL=0  +MOVJ EC01466
COMM ARCON
COMM SMOVL C01467 BC01467 V=10.0  +MOVJ EC01467
COMM SMOVL C01468 BC01468 V=10.0  +MOVJ EC01468
COMM SMOVL C01469 BC01469 V=10.0  +MOVJ EC01469
COMM ARCON
COMM SMOVL C01470 BC01470 V=11.7  +MOVJ EC01470
COMM ARCON
COMM SMOVL C01471 BC01471 V=11.7  +MOVJ EC01471
COMM ARCOF
COMM SMOVL C01472 BC01472 V=800.0  +MOVJ EC01472
COMM SMOVL C01473 BC01473 V=1000.0  +MOVJ EC01473
COMM SFTOF3D
COMM 'EndPath W3493
COMM MOVJ C01474 BC01474 VJ=100.00  +MOVJ EC01474 VJ=100.00
COMM MOVJ C01475 BC01475 VJ=100.00  +MOVJ EC01475 VJ=100.00
COMM '16
COMM 'Path W3491
COMM SFTOF3D
COMM SFTON3D P080
COMM MOVJ C01476 BC01476 VJ=100.00  +MOVJ EC01476 VJ=100.00
COMM SMOVL C01477 BC01477 V=800.0  +MOVJ EC01477
COMM SMOVL C01478 BC01478 V=150.0 PL=0  +MOVJ EC01478
COMM ARCON
COMM SMOVL C01479 BC01479 V=10.0  +MOVJ EC01479
COMM SMOVL C01480 BC01480 V=10.0  +MOVJ EC01480
COMM ARCOF
COMM SMOVL C01481 BC01481 V=800.0  +MOVJ EC01481
COMM SMOVL C01482 BC01482 V=1000.0  +MOVJ EC01482
COMM SFTOF3D
COMM 'EndPath W3491
COMM MOVJ C01483 BC01483 VJ=100.00  +MOVJ EC01483 VJ=100.00
COMM 'Path W3492
COMM SFTOF3D
COMM SFTON3D P080
COMM MOVJ C01484 BC01484 VJ=100.00  +MOVJ EC01484 VJ=100.00
COMM SMOVL C01485 BC01485 V=800.0  +MOVJ EC01485
COMM SMOVL C01486 BC01486 V=150.0 PL=0  +MOVJ EC01486
COMM ARCON
COMM SMOVL C01487 BC01487 V=10.0  +MOVJ EC01487
COMM ARCOF
COMM SMOVL C01488 BC01488 V=800.0  +MOVJ EC01488
COMM SMOVL C01489 BC01489 V=1000.0  +MOVJ EC01489
COMM SFTOF3D
COMM 'EndPath W3492
COMM MOVJ C01490 BC01490 VJ=100.00  +MOVJ EC01490 VJ=100.00
COMM MOVJ C01491 BC01491 VJ=100.00  +MOVJ EC01491 VJ=100.00
COMM 'Path W3493
COMM SFTOF3D
COMM SFTON3D P080
COMM MOVJ C01492 BC01492 VJ=100.00  +MOVJ EC01492 VJ=100.00
COMM SMOVL C01493 BC01493 V=800.0  +MOVJ EC01493
COMM SMOVL C01494 BC01494 V=150.0 PL=0  +MOVJ EC01494
COMM ARCON
COMM SMOVL C01495 BC01495 V=10.0  +MOVJ EC01495
COMM SMOVL C01496 BC01496 V=10.0  +MOVJ EC01496
COMM SMOVL C01497 BC01497 V=10.0  +MOVJ EC01497
COMM ARCON
COMM SMOVL C01498 BC01498 V=11.7  +MOVJ EC01498
COMM ARCON
COMM SMOVL C01499 BC01499 V=11.7  +MOVJ EC01499
COMM ARCOF
COMM SMOVL C01500 BC01500 V=800.0  +MOVJ EC01500
COMM SMOVL C01501 BC01501 V=1000.0  +MOVJ EC01501
COMM SFTOF3D
COMM 'EndPath W3493
COMM MOVJ C01502 BC01502 VJ=100.00  +MOVJ EC01502 VJ=100.00
COMM MOVJ C01503 BC01503 VJ=100.00  +MOVJ EC01503 VJ=100.00
COMM '17
COMM 'Path W3494
COMM SFTOF3D
COMM SFTON3D P027
COMM MOVJ C01504 BC01504 VJ=100.00  +MOVJ EC01504 VJ=100.00
COMM SMOVL C01505 BC01505 V=800.0  +MOVJ EC01505
COMM SMOVL C01506 BC01506 V=150.0 PL=0  +MOVJ EC01506
COMM ARCON
COMM SMOVL C01507 BC01507 V=10.0  +MOVJ EC01507
COMM ARCOF
COMM SMOVL C01508 BC01508 V=800.0  +MOVJ EC01508
COMM SMOVL C01509 BC01509 V=1000.0  +MOVJ EC01509
COMM SFTOF3D
COMM 'EndPath W3494
COMM 'Path W3495
COMM SFTOF3D
COMM SFTON3D P027
COMM MOVJ C01510 BC01510 VJ=100.00  +MOVJ EC01510 VJ=100.00
COMM SMOVL C01511 BC01511 V=800.0  +MOVJ EC01511
COMM SMOVL C01512 BC01512 V=150.0 PL=0  +MOVJ EC01512
COMM ARCON
COMM SMOVL C01513 BC01513 V=10.8  +MOVJ EC01513
COMM ARCOF
COMM SMOVL C01514 BC01514 V=800.0  +MOVJ EC01514
COMM SMOVL C01515 BC01515 V=1000.0  +MOVJ EC01515
COMM SFTOF3D
COMM 'EndPath W3495
COMM 'Path W3496
COMM SFTOF3D
COMM SFTON3D P027
COMM MOVJ C01516 BC01516 VJ=100.00  +MOVJ EC01516 VJ=100.00
COMM SFTOF3D
COMM 'EndPath W3496
COMM MOVJ C01517 BC01517 VJ=100.00  +MOVJ EC01517 VJ=100.00
COMM MOVJ C01518 BC01518 VJ=100.00  +MOVJ EC01518 VJ=100.00
COMM MOVJ C01519 BC01519 VJ=100.00  +MOVJ EC01519 VJ=100.00
COMM '18
COMM 'Path W3497
COMM SFTOF3D
COMM SFTON3D P024
COMM MOVJ C01520 BC01520 VJ=100.00  +MOVJ EC01520 VJ=100.00
COMM SMOVL C01521 BC01521 V=800.0  +MOVJ EC01521
COMM SMOVL C01522 BC01522 V=150.0 PL=0  +MOVJ EC01522
COMM ARCON
COMM SMOVL C01523 BC01523 V=9.2  +MOVJ EC01523
COMM SMOVL C01524 BC01524 V=9.2  +MOVJ EC01524
COMM SMOVL C01525 BC01525 V=9.2  +MOVJ EC01525
COMM SMOVL C01526 BC01526 V=9.2  +MOVJ EC01526
COMM ARCOF
COMM SMOVL C01527 BC01527 V=800.0  +MOVJ EC01527
COMM SMOVL C01528 BC01528 V=1000.0  +MOVJ EC01528
COMM SFTOF3D
COMM 'EndPath W3497
COMM '
COMM 'Path W4855
COMM SFTOF3D
COMM SFTON3D P071
COMM MOVJ C01529 BC01529 VJ=100.00  +MOVJ EC01529 VJ=100.00
COMM SMOVL C01530 BC01530 V=800.0  +MOVJ EC01530
COMM MACRO1 MJ#(0) ARGF9
COMM SMOVL C01531 BC01531 V=150.0 PL=0  +MOVJ EC01531
COMM ARCON
COMM SMOVL C01532 BC01532 V=8.8  +MOVJ EC01532
COMM SFTON3D P072
COMM SMOVL C01533 BC01533 V=8.8  +MOVJ EC01533
COMM SMOVL C01534 BC01534 V=8.8  +MOVJ EC01534
COMM ARCOF
COMM SMOVL C01535 BC01535 V=166.7  +MOVJ EC01535
COMM SMOVL C01536 BC01536 V=800.0  +MOVJ EC01536
COMM SMOVL C01537 BC01537 V=800.0  +MOVJ EC01537
COMM SMOVL C01538 BC01538 V=800.0  +MOVJ EC01538
COMM SFTON3D P072
COMM SMOVL C01539 BC01539 V=166.7 PL=0  +MOVJ EC01539
COMM ARCON
COMM SMOVL C01540 BC01540 V=8.8  +MOVJ EC01540
COMM SMOVL C01541 BC01541 V=8.8  +MOVJ EC01541
COMM SMOVL C01542 BC01542 V=8.8  +MOVJ EC01542
COMM SMOVL C01543 BC01543 V=8.8  +MOVJ EC01543
COMM ARCOF
COMM MOVL C01544 BC01544 V=166.7  +MOVJ EC01544 VJ=0.78
COMM SMOVL C01545 BC01545 V=1000.0  +MOVJ EC01545
COMM SFTOF3D
COMM 'EndPath W4855
COMM '
COMM '
COMM MOVJ C01546 BC01546 VJ=100.00  +MOVJ EC01546 VJ=100.00
COMM '19
COMM MOVJ C01547 BC01547 VJ=100.00  +MOVJ EC01547 VJ=100.00
COMM 'Path W3499
COMM SFTOF3D
COMM SFTON3D P023
COMM MOVJ C01548 BC01548 VJ=100.00  +MOVJ EC01548 VJ=100.00
COMM SMOVL C01549 BC01549 V=800.0  +MOVJ EC01549
COMM SMOVL C01550 BC01550 V=150.0 PL=0  +MOVJ EC01550
COMM MACRO1 MJ#(0) ARGF6
COMM ARCON
COMM SWVON WEV#(66)
COMM SMOVL C01551 BC01551 V=7.5  +MOVJ EC01551
COMM SMOVL C01552 BC01552 V=7.5  +MOVJ EC01552
COMM SMOVL C01553 BC01553 V=7.5  +MOVJ EC01553
COMM ARCOF
COMM SWVOF
COMM SMOVL C01554 BC01554 V=800.0  +MOVJ EC01554
COMM SMOVL C01555 BC01555 V=1000.0  +MOVJ EC01555
COMM SFTOF3D
COMM 'EndPath W3499
COMM MOVJ C01556 BC01556 VJ=100.00  +MOVJ EC01556 VJ=100.00
COMM 'Path W3500
COMM SFTOF3D
COMM SFTON3D P034
COMM MOVJ C01557 BC01557 VJ=100.00  +MOVJ EC01557 VJ=100.00
COMM SMOVL C01558 BC01558 V=800.0  +MOVJ EC01558
COMM MACRO1 MJ#(0) ARGF9
COMM SMOVL C01559 BC01559 V=150.0 PL=0  +MOVJ EC01559
COMM ARCON
COMM SMOVL C01560 BC01560 V=8.3  +MOVJ EC01560
COMM SFTON3D P050
COMM SMOVL C01561 BC01561 V=8.3  +MOVJ EC01561
COMM SMOVL C01562 BC01562 V=8.3  +MOVJ EC01562
COMM ARCOF
COMM SMOVL C01563 BC01563 V=800.0  +MOVJ EC01563
COMM SMOVL C01564 BC01564 V=1000.0  +MOVJ EC01564
COMM SFTOF3D
COMM 'EndPath W3500
COMM 'Path W3501
COMM SFTOF3D
COMM SFTON3D P051
COMM MOVJ C01565 BC01565 VJ=100.00  +MOVJ EC01565 VJ=100.00
COMM SMOVL C01566 BC01566 V=800.0  +MOVJ EC01566
COMM SMOVL C01567 BC01567 V=150.0 PL=0  +MOVJ EC01567
COMM ARCON
COMM SWVON WEV#(60)
COMM SMOVL C01568 BC01568 V=7.5  +MOVJ EC01568
COMM SMOVL C01569 BC01569 V=7.5  +MOVJ EC01569
COMM SMOVL C01570 BC01570 V=7.5  +MOVJ EC01570
COMM ARCOF
COMM SWVOF
COMM SMOVL C01571 BC01571 V=800.0  +MOVJ EC01571
COMM SMOVL C01572 BC01572 V=1000.0  +MOVJ EC01572
COMM SFTOF3D
COMM 'EndPath W3501
COMM MOVJ C01573 BC01573 VJ=100.00  +MOVJ EC01573 VJ=100.00
COMM '20
COMM MOVJ C01574 BC01574 VJ=100.00  +MOVJ EC01574 VJ=100.00
COMM MOVJ C01575 BC01575 VJ=100.00  +MOVJ EC01575 VJ=100.00
COMM 'offset 5mm
COMM 'Path W3500
COMM SFTOF3D
COMM SFTON3D P032
COMM MOVJ C01576 BC01576 VJ=100.00  +MOVJ EC01576 VJ=100.00
COMM SMOVL C01577 BC01577 V=800.0  +MOVJ EC01577
COMM SMOVL C01578 BC01578 V=150.0 PL=0  +MOVJ EC01578
COMM ARCON
COMM SMOVL C01579 BC01579 V=9.2  +MOVJ EC01579
COMM ARCOF
COMM SMOVL C01580 BC01580 V=800.0  +MOVJ EC01580
COMM SMOVL C01581 BC01581 V=1000.0  +MOVJ EC01581
COMM SFTOF3D
COMM 'EndPath W3500
COMM SFTOF3D
COMM 'EndPath W3502
COMM 'offset 5mm
COMM 'Path W3503
COMM SFTOF3D
COMM SFTON3D P032
COMM MOVJ C01582 BC01582 VJ=100.00  +MOVJ EC01582 VJ=100.00
COMM SMOVL C01583 BC01583 V=800.0  +MOVJ EC01583
COMM SMOVL C01584 BC01584 V=150.0 PL=0  +MOVJ EC01584
COMM ARCON
COMM SMOVL C01585 BC01585 V=10.0  +MOVJ EC01585
COMM ARCOF
COMM SMOVL C01586 BC01586 V=800.0  +MOVJ EC01586
COMM SMOVL C01587 BC01587 V=1000.0  +MOVJ EC01587
COMM SFTOF3D
COMM 'EndPath W3503
COMM MOVJ C01588 BC01588 VJ=100.00  +MOVJ EC01588 VJ=100.00
COMM 'Path W3504
COMM SFTOF3D
COMM SFTON3D P032
COMM MOVJ C01589 BC01589 VJ=100.00  +MOVJ EC01589 VJ=100.00
COMM SMOVL C01590 BC01590 V=800.0  +MOVJ EC01590
COMM SMOVL C01591 BC01591 V=150.0 PL=0  +MOVJ EC01591
COMM ARCON
COMM SMOVL C01592 BC01592 V=11.7  +MOVJ EC01592
COMM SMOVL C01593 BC01593 V=11.7  +MOVJ EC01593
COMM ARCOF
COMM SMOVL C01594 BC01594 V=800.0  +MOVJ EC01594
COMM SMOVL C01595 BC01595 V=1000.0  +MOVJ EC01595
COMM SFTOF3D
COMM 'EndPath W3504
COMM MOVJ C01596 BC01596 VJ=100.00  +MOVJ EC01596 VJ=100.00
COMM '21
COMM MOVJ C01597 BC01597 VJ=100.00  +MOVJ EC01597 VJ=100.00
COMM 'Path W3505
COMM SFTOF3D
COMM SFTON3D P021
COMM MOVJ C01598 BC01598 VJ=100.00  +MOVJ EC01598 VJ=100.00
COMM SMOVL C01599 BC01599 V=800.0  +MOVJ EC01599
COMM SMOVL C01600 BC01600 V=150.0 PL=0  +MOVJ EC01600
COMM ARCON
COMM SFTON3D P022
COMM SMOVL C01601 BC01601 V=10.8  +MOVJ EC01601
COMM SMOVL C01602 BC01602 V=11.7  +MOVJ EC01602
COMM ARCOF
COMM SMOVL C01603 BC01603 V=800.0  +MOVJ EC01603
COMM SMOVL C01604 BC01604 V=1000.0  +MOVJ EC01604
COMM SFTOF3D
COMM 'EndPath W3505
COMM MOVJ C01605 BC01605 VJ=100.00  +MOVJ EC01605 VJ=100.00
COMM 'Path W3506
COMM SFTOF3D
COMM SFTON3D P095
COMM MOVJ C01606 BC01606 VJ=100.00  +MOVJ EC01606 VJ=100.00
COMM SMOVL C01607 BC01607 V=800.0  +MOVJ EC01607
COMM SMOVL C01608 BC01608 V=150.0 PL=0  +MOVJ EC01608
COMM MACRO1 MJ#(0) ARGF14
COMM ARCON
COMM SMOVL C01609 BC01609 V=10.0  +MOVJ EC01609
COMM SMOVL C01610 BC01610 V=10.0  +MOVJ EC01610
COMM SMOVL C01611 BC01611 V=10.0  +MOVJ EC01611
COMM ARCOF
COMM SMOVL C01612 BC01612 V=800.0  +MOVJ EC01612
COMM SMOVL C01613 BC01613 V=1000.0  +MOVJ EC01613
COMM SFTOF3D
COMM 'EndPath W3506
COMM 'Path W3507
COMM SFTOF3D
COMM SFTON3D P096
COMM MOVJ C01614 BC01614 VJ=100.00  +MOVJ EC01614 VJ=100.00
COMM SMOVL C01615 BC01615 V=800.0  +MOVJ EC01615
COMM SMOVL C01616 BC01616 V=150.0 PL=0  +MOVJ EC01616
COMM ARCON
COMM SMOVL C01617 BC01617 V=10.0  +MOVJ EC01617
COMM SMOVL C01618 BC01618 V=10.0  +MOVJ EC01618
COMM ARCOF
COMM SMOVL C01619 BC01619 V=800.0  +MOVJ EC01619
COMM SMOVL C01620 BC01620 V=1000.0  +MOVJ EC01620
COMM SFTOF3D
COMM 'EndPath W3507
COMM MOVJ C01621 BC01621 VJ=100.00  +MOVJ EC01621 VJ=100.00
COMM MOVJ C01622 BC01622 VJ=100.00  +MOVJ EC01622 VJ=100.00
COMM 'Path W4856
COMM SFTOF3D
COMM SFTON3D P071
COMM MOVJ C01623 BC01623 VJ=100.00  +MOVJ EC01623 VJ=100.00
COMM SMOVL C01624 BC01624 V=800.0  +MOVJ EC01624
COMM SMOVL C01625 BC01625 V=150.0 PL=0  +MOVJ EC01625
COMM ARCON
COMM SMOVL C01626 BC01626 V=8.3  +MOVJ EC01626
COMM SFTON3D P073
COMM SMOVL C01627 BC01627 V=8.3  +MOVJ EC01627
COMM SMOVL C01628 BC01628 V=8.3  +MOVJ EC01628
COMM ARCOF
COMM SMOVL C01629 BC01629 V=800.0  +MOVJ EC01629
COMM SMOVL C01630 BC01630 V=1000.0  +MOVJ EC01630
COMM SFTOF3D
COMM 'EndPath W4856
COMM MOVJ C01631 BC01631 VJ=100.00  +MOVJ EC01631 VJ=100.00
COMM MOVJ C01632 BC01632 VJ=50.00  +MOVJ EC01632 VJ=0.78
COMM MOVJ C01633 BC01633 VJ=100.00  +MOVJ EC01633 VJ=50.00
COMM SFTON3D P080
COMM SMOVL C01634 BC01634 V=800.0  +MOVJ EC01634
COMM SMOVL C01635 BC01635 V=150.0 PL=0  +MOVJ EC01635
COMM ARCON
COMM SMOVL C01636 BC01636 V=8.3  +MOVJ EC01636
COMM SMOVL C01637 BC01637 V=8.3  +MOVJ EC01637
COMM SMOVC C01638 BC01638 V=8.3  +MOVJ EC01638
COMM ARCOF
COMM SMOVL C01639 BC01639 V=800.0  +MOVJ EC01639
COMM SFTOF3D
COMM SMOVL C01640 BC01640 V=1000.0  +MOVJ EC01640
COMM MOVJ C01641 BC01641 VJ=100.00  +MOVJ EC01641 VJ=100.00
COMM MOVJ C01642 BC01642 VJ=100.00  +MOVJ EC01642 VJ=100.00
COMM MOVJ C01643 BC01643 VJ=100.00  +MOVJ EC01643 VJ=100.00
COMM MOVJ C01644 BC01644 VJ=100.00  +MOVJ EC01644 VJ=100.00
COMM SFTON3D P081
COMM SMOVL C01645 BC01645 V=666.7  +MOVJ EC01645
COMM SMOVL C01646 BC01646 V=166.7 PL=0  +MOVJ EC01646
COMM ARCON
COMM SMOVL C01647 BC01647 V=8.3  +MOVJ EC01647
COMM SMOVL C01648 BC01648 V=8.3  +MOVJ EC01648
COMM SMOVL C01649 BC01649 V=8.3  +MOVJ EC01649
COMM ARCOF
COMM SMOVL C01650 BC01650 V=333.3  +MOVJ EC01650
COMM SFTOF3D
COMM MOVL C01651 BC01651 V=1000.0  +MOVJ EC01651 VJ=100.00
COMM MOVJ C01652 BC01652 VJ=100.00  +MOVJ EC01652 VJ=100.00
COMM MOVJ C01653 BC01653 VJ=100.00  +MOVJ EC01653 VJ=100.00
COMM 'cut_wire_dol
COMM 'cut_wire_dol
COMM 'cut_wire_dol
COMM CALL JOB:CLEAN-R1_KM_NEW
MOVJ C01654 BC01654 VJ=100.00  +MOVJ EC01654 VJ=100.00
MOVJ C01655 BC01655 VJ=100.00  +MOVJ EC01655 VJ=100.00
MOVJ C01656 BC01656 VJ=100.00  +MOVJ EC01656 VJ=100.00
'Path S4011
SFTOF3D
MOVJ C01657 BC01657 VJ=100.00  +MOVJ EC01657 VJ=100.00
MOVL C01658 BC01658 V=666.7  +MOVJ EC01658 VJ=100.00
SMOVL C01659 BC01659 V=166.7  +MOVJ EC01659
SREFP 3 C01660 BC01660  +REFP EC01660
CALL JOB:SEARCH-R1-S13D
SET P049 P006
SFTON3D P049
SMOVL C01661 BC01661 V=166.7  +MOVJ EC01661
SMOVL C01662 BC01662 V=166.7  +MOVJ EC01662
SREFP 3 C01663 BC01663  +REFP EC01663
CALL JOB:SEARCH-R1-S13D
SET P049 P006
SFTON3D P049
SMOVL C01664 BC01664 V=166.7  +MOVJ EC01664
MOVL C01665 BC01665 V=1000.0  +MOVJ EC01665 VJ=100.00
'EndPath S4011
'Path S4010
SFTOF3D
MOVJ C01666 BC01666 VJ=100.00  +MOVJ EC01666 VJ=100.00
SMOVL C01667 BC01667 V=666.7  +MOVJ EC01667
SMOVL C01668 BC01668 V=166.7  +MOVJ EC01668
SREFP 3 C01669 BC01669  +REFP EC01669
CALL JOB:SEARCH-R1-S13D
SET P048 P006
SFTON3D P048
SMOVL C01670 BC01670 V=166.7  +MOVJ EC01670
SMOVL C01671 BC01671 V=166.7  +MOVJ EC01671
SREFP 3 C01672 BC01672  +REFP EC01672
CALL JOB:SEARCH-R1-S13D
SET P048 P006
SFTON3D P048
SMOVL C01673 BC01673 V=233.3  +MOVJ EC01673
MOVL C01674 BC01674 V=1000.0  +MOVJ EC01674 VJ=100.00
'EndPath S4010
'Path S4009
SFTOF3D
MOVJ C01675 BC01675 VJ=100.00  +MOVJ EC01675 VJ=100.00
MOVL C01676 BC01676 V=666.7  +MOVJ EC01676 VJ=100.00
SMOVL C01677 BC01677 V=166.7  +MOVJ EC01677
SREFP 3 C01678 BC01678  +REFP EC01678
CALL JOB:SEARCH-R1-S13D
SET P047 P006
SFTON3D P047
SMOVL C01679 BC01679 V=166.7  +MOVJ EC01679
SMOVL C01680 BC01680 V=166.7  +MOVJ EC01680
SREFP 3 C01681 BC01681  +REFP EC01681
CALL JOB:SEARCH-R1-S13D
SET P047 P006
SFTON3D P047
SMOVL C01682 BC01682 V=166.7  +MOVJ EC01682
MOVL C01683 BC01683 V=1000.0  +MOVJ EC01683 VJ=100.00
'EndPath S4009
MOVJ C01684 BC01684 VJ=100.00  +MOVJ EC01684 VJ=100.00
'Path S4008
SFTOF3D
MOVJ C01685 BC01685 VJ=100.00  +MOVJ EC01685 VJ=100.00
MOVL C01686 BC01686 V=666.7  +MOVJ EC01686 VJ=100.00
SMOVL C01687 BC01687 V=166.7  +MOVJ EC01687
SREFP 3 C01688 BC01688  +REFP EC01688
CALL JOB:SEARCH-R1-S13D
SET P046 P006
SFTON3D P046
SMOVL C01689 BC01689 V=166.7  +MOVJ EC01689
SMOVL C01690 BC01690 V=166.7  +MOVJ EC01690
SREFP 3 C01691 BC01691  +REFP EC01691
CALL JOB:SEARCH-R1-S13D
SET P046 P006
SFTON3D P046
SMOVL C01692 BC01692 V=166.7  +MOVJ EC01692
MOVL C01693 BC01693 V=1000.0  +MOVJ EC01693 VJ=100.00
'EndPath S4008
'Path S4007
SFTOF3D
MOVJ C01694 BC01694 VJ=100.00  +MOVJ EC01694 VJ=100.00
MOVL C01695 BC01695 V=666.7  +MOVJ EC01695 VJ=100.00
SMOVL C01696 BC01696 V=166.7  +MOVJ EC01696
SREFP 3 C01697 BC01697  +REFP EC01697
CALL JOB:SEARCH-R1-S13D
SET P045 P006
SFTON3D P045
SMOVL C01698 BC01698 V=166.7  +MOVJ EC01698
SMOVL C01699 BC01699 V=166.7  +MOVJ EC01699
SMOVL C01700 BC01700 V=166.7  +MOVJ EC01700
SREFP 3 C01701 BC01701  +REFP EC01701
CALL JOB:SEARCH-R1-S13D
SET P045 P006
SFTON3D P045
SMOVL C01702 BC01702 V=166.7  +MOVJ EC01702
MOVL C01703 BC01703 V=1000.0  +MOVJ EC01703 VJ=100.00
'EndPath S4007
'Path S3506
SFTOF3D
MOVJ C01704 BC01704 VJ=100.00  +MOVJ EC01704 VJ=100.00
MOVL C01705 BC01705 V=666.7  +MOVJ EC01705 VJ=100.00
SMOVL C01706 BC01706 V=166.7  +MOVJ EC01706
SREFP 3 C01707 BC01707  +REFP EC01707
CALL JOB:SEARCH-R1-S13D
SET P044 P006
SFTON3D P044
SMOVL C01708 BC01708 V=166.7  +MOVJ EC01708
SMOVL C01709 BC01709 V=166.7  +MOVJ EC01709
SREFP 3 C01710 BC01710  +REFP EC01710
CALL JOB:SEARCH-R1-S13D
SET P044 P006
SFTON3D P044
SMOVL C01711 BC01711 V=166.7  +MOVJ EC01711
MOVL C01712 BC01712 V=1000.0  +MOVJ EC01712 VJ=100.00
'EndPath S3506
MOVJ C01713 BC01713 VJ=100.00  +MOVJ EC01713 VJ=100.00
MOVJ C01714 BC01714 VJ=100.00  +MOVJ EC01714 VJ=100.00
MOVJ C01715 BC01715 VJ=100.00  +MOVJ EC01715 VJ=100.00
MOVJ C01716 BC01716 VJ=100.00  +MOVJ EC01716 VJ=100.00
MOVJ C01717 BC01717 VJ=100.00  +MOVJ EC01717 VJ=100.00
'Path S4006
SFTOF3D
MOVJ C01718 BC01718 VJ=100.00  +MOVJ EC01718 VJ=100.00
MOVL C01719 BC01719 V=666.7  +MOVJ EC01719 VJ=100.00
SMOVL C01720 BC01720 V=166.7  +MOVJ EC01720
SREFP 3 C01721 BC01721  +REFP EC01721
CALL JOB:SEARCH-R1-S13D
SET P043 P006
SFTON3D P043
SMOVL C01722 BC01722 V=166.7  +MOVJ EC01722
SMOVL C01723 BC01723 V=166.7  +MOVJ EC01723
SMOVL C01724 BC01724 V=166.7  +MOVJ EC01724
SREFP 3 C01725 BC01725  +REFP EC01725
CALL JOB:SEARCH-R1-S13D
SET P043 P006
SFTON3D P043
SMOVL C01726 BC01726 V=166.7  +MOVJ EC01726
MOVL C01727 BC01727 V=1000.0  +MOVJ EC01727 VJ=100.00
'EndPath S4006
'Path S4005
SFTOF3D
MOVJ C01728 BC01728 VJ=100.00  +MOVJ EC01728 VJ=100.00
MOVL C01729 BC01729 V=800.0  +MOVJ EC01729 VJ=100.00
SMOVL C01730 BC01730 V=166.7  +MOVJ EC01730
SREFP 3 C01731 BC01731  +REFP EC01731
CALL JOB:SEARCH-R1-S13D
SET P042 P006
SFTON3D P042
SMOVL C01732 BC01732 V=166.7  +MOVJ EC01732
SMOVL C01733 BC01733 V=166.7  +MOVJ EC01733
SREFP 3 C01734 BC01734  +REFP EC01734
CALL JOB:SEARCH-R1-S13D
SET P042 P006
SFTON3D P042
SMOVL C01735 BC01735 V=166.7  +MOVJ EC01735
MOVL C01736 BC01736 V=1000.0  +MOVJ EC01736 VJ=100.00
'EndPath S4005
'Path S4004
SFTOF3D
MOVJ C01737 BC01737 VJ=100.00  +MOVJ EC01737 VJ=100.00
MOVL C01738 BC01738 V=800.0  +MOVJ EC01738 VJ=100.00
SMOVL C01739 BC01739 V=166.7  +MOVJ EC01739
SMOVL C01740 BC01740 V=166.7  +MOVJ EC01740
SREFP 3 C01741 BC01741  +REFP EC01741
CALL JOB:SEARCH-R1-S13D
SET P041 P006
SFTON3D P041
SMOVL C01742 BC01742 V=166.7  +MOVJ EC01742
SMOVL C01743 BC01743 V=166.7  +MOVJ EC01743
SREFP 3 C01744 BC01744  +REFP EC01744
CALL JOB:SEARCH-R1-S13D
SET P041 P006
SFTON3D P041
SMOVL C01745 BC01745 V=166.7  +MOVJ EC01745
SREFP 3 C01746 BC01746  +REFP EC01746
CALL JOB:SEARCH-R1-S13D
SET P041 P006
SFTON3D P041
SMOVL C01747 BC01747 V=166.7  +MOVJ EC01747
MOVL C01748 BC01748 V=1000.0  +MOVJ EC01748 VJ=100.00
'EndPath S4004
'Path S4003
SFTOF3D
MOVJ C01749 BC01749 VJ=100.00  +MOVJ EC01749 VJ=100.00
MOVL C01750 BC01750 V=800.0  +MOVJ EC01750 VJ=100.00
SMOVL C01751 BC01751 V=166.7  +MOVJ EC01751
SREFP 3 C01752 BC01752  +REFP EC01752
CALL JOB:SEARCH-R1-S13D
SET P040 P006
SFTON3D P040
SMOVL C01753 BC01753 V=250.0  +MOVJ EC01753
SMOVL C01754 BC01754 V=250.0  +MOVJ EC01754
SMOVL C01755 BC01755 V=166.7  +MOVJ EC01755
SREFP 3 C01756 BC01756  +REFP EC01756
CALL JOB:SEARCH-R1-S13D
SET P040 P006
SFTON3D P040
SMOVL C01757 BC01757 V=166.7  +MOVJ EC01757
SMOVL C01758 BC01758 V=166.7  +MOVJ EC01758
SREFP 3 C01759 BC01759  +REFP EC01759
CALL JOB:SEARCH-R1-S13D
SET P040 P006
SFTON3D P040
SMOVL C01760 BC01760 V=166.7  +MOVJ EC01760
MOVL C01761 BC01761 V=1000.0  +MOVJ EC01761 VJ=100.00
'EndPath S4003
'Path W4012
SFTOF3D
SFTON3D P040
MOVJ C01762 BC01762 VJ=100.00  +MOVJ EC01762 VJ=100.00
SMOVL C01763 BC01763 V=800.0  +MOVJ EC01763
SMOVL C01764 BC01764 V=150.0 PL=0  +MOVJ EC01764
ARCON
SMOVL C01765 BC01765 V=11.7  +MOVJ EC01765
ARCOF
SMOVL C01766 BC01766 V=800.0  +MOVJ EC01766
SMOVL C01767 BC01767 V=1000.0  +MOVJ EC01767
SFTOF3D
'EndPath W4012
'Path W4013
SFTOF3D
SFTON3D P040
MOVJ C01768 BC01768 VJ=100.00  +MOVJ EC01768 VJ=100.00
SMOVL C01769 BC01769 V=800.0  +MOVJ EC01769
SMOVL C01770 BC01770 V=150.0 PL=0  +MOVJ EC01770
ARCON
SMOVL C01771 BC01771 V=10.0  +MOVJ EC01771
ARCOF
SMOVL C01772 BC01772 V=800.0  +MOVJ EC01772
